        FuUnicodeCodepointCaseConvert := 43900;
        RETURN;
    5037:
        FuUnicodeCodepointCaseConvert := 43901;
        RETURN;
    5038:
        FuUnicodeCodepointCaseConvert := 43902;
        RETURN;
    5039:
        FuUnicodeCodepointCaseConvert := 43903;
        RETURN;
    5040:
        FuUnicodeCodepointCaseConvert := 43904;
        RETURN;
    5041:
        FuUnicodeCodepointCaseConvert := 43905;
        RETURN;
    5042:
        FuUnicodeCodepointCaseConvert := 43906;
        RETURN;
    5043:
        FuUnicodeCodepointCaseConvert := 43907;
        RETURN;
    5044:
        FuUnicodeCodepointCaseConvert := 43908;
        RETURN;
    5045:
        FuUnicodeCodepointCaseConvert := 43909;
        RETURN;
    5046:
        FuUnicodeCodepointCaseConvert := 43910;
        RETURN;
    5047:
        FuUnicodeCodepointCaseConvert := 43911;
        RETURN;
    5048:
        FuUnicodeCodepointCaseConvert := 43912;
        RETURN;
    5049:
        FuUnicodeCodepointCaseConvert := 43913;
        RETURN;
    5050:
        FuUnicodeCodepointCaseConvert := 43914;
        RETURN;
    5051:
        FuUnicodeCodepointCaseConvert := 43915;
        RETURN;
    5052:
        FuUnicodeCodepointCaseConvert := 43916;
        RETURN;
    5053:
        FuUnicodeCodepointCaseConvert := 43917;
        RETURN;
    5054:
        FuUnicodeCodepointCaseConvert := 43918;
        RETURN;
    5055:
        FuUnicodeCodepointCaseConvert := 43919;
        RETURN;
    5056:
        FuUnicodeCodepointCaseConvert := 43920;
        RETURN;
    5057:
        FuUnicodeCodepointCaseConvert := 43921;
        RETURN;
    5058:
        FuUnicodeCodepointCaseConvert := 43922;
        RETURN;
    5059:
        FuUnicodeCodepointCaseConvert := 43923;
        RETURN;
    5060:
        FuUnicodeCodepointCaseConvert := 43924;
        RETURN;
    5061:
        FuUnicodeCodepointCaseConvert := 43925;
        RETURN;
    5062:
        FuUnicodeCodepointCaseConvert := 43926;
        RETURN;
    5063:
        FuUnicodeCodepointCaseConvert := 43927;
        RETURN;
    5064:
        FuUnicodeCodepointCaseConvert := 43928;
        RETURN;
    5065:
        FuUnicodeCodepointCaseConvert := 43929;
        RETURN;
    5066:
        FuUnicodeCodepointCaseConvert := 43930;
        RETURN;
    5067:
        FuUnicodeCodepointCaseConvert := 43931;
        RETURN;
    5068:
        FuUnicodeCodepointCaseConvert := 43932;
        RETURN;
    5069:
        FuUnicodeCodepointCaseConvert := 43933;
        RETURN;
    5070:
        FuUnicodeCodepointCaseConvert := 43934;
        RETURN;
    5071:
        FuUnicodeCodepointCaseConvert := 43935;
        RETURN;
    5072:
        FuUnicodeCodepointCaseConvert := 43936;
        RETURN;
    5073:
        FuUnicodeCodepointCaseConvert := 43937;
        RETURN;
    5074:
        FuUnicodeCodepointCaseConvert := 43938;
        RETURN;
    5075:
        FuUnicodeCodepointCaseConvert := 43939;
        RETURN;
    5076:
        FuUnicodeCodepointCaseConvert := 43940;
        RETURN;
    5077:
        FuUnicodeCodepointCaseConvert := 43941;
        RETURN;
    5078:
        FuUnicodeCodepointCaseConvert := 43942;
        RETURN;
    5079:
        FuUnicodeCodepointCaseConvert := 43943;
        RETURN;
    5080:
        FuUnicodeCodepointCaseConvert := 43944;
        RETURN;
    5081:
        FuUnicodeCodepointCaseConvert := 43945;
        RETURN;
    5082:
        FuUnicodeCodepointCaseConvert := 43946;
        RETURN;
    5083:
        FuUnicodeCodepointCaseConvert := 43947;
        RETURN;
    5084:
        FuUnicodeCodepointCaseConvert := 43948;
        RETURN;
    5085:
        FuUnicodeCodepointCaseConvert := 43949;
        RETURN;
    5086:
        FuUnicodeCodepointCaseConvert := 43950;
        RETURN;
    5087:
        FuUnicodeCodepointCaseConvert := 43951;
        RETURN;
    5088:
        FuUnicodeCodepointCaseConvert := 43952;
        RETURN;
    5089:
        FuUnicodeCodepointCaseConvert := 43953;
        RETURN;
    5090:
        FuUnicodeCodepointCaseConvert := 43954;
        RETURN;
    5091:
        FuUnicodeCodepointCaseConvert := 43955;
        RETURN;
    5092:
        FuUnicodeCodepointCaseConvert := 43956;
        RETURN;
    5093:
        FuUnicodeCodepointCaseConvert := 43957;
        RETURN;
    5094:
        FuUnicodeCodepointCaseConvert := 43958;
        RETURN;
    5095:
        FuUnicodeCodepointCaseConvert := 43959;
        RETURN;
    5096:
        FuUnicodeCodepointCaseConvert := 43960;
        RETURN;
    5097:
        FuUnicodeCodepointCaseConvert := 43961;
        RETURN;
    5098:
        FuUnicodeCodepointCaseConvert := 43962;
        RETURN;
    5099:
        FuUnicodeCodepointCaseConvert := 43963;
        RETURN;
    5100:
        FuUnicodeCodepointCaseConvert := 43964;
        RETURN;
    5101:
        FuUnicodeCodepointCaseConvert := 43965;
        RETURN;
    5102:
        FuUnicodeCodepointCaseConvert := 43966;
        RETURN;
    5103:
        FuUnicodeCodepointCaseConvert := 43967;
        RETURN;
    5104:
        FuUnicodeCodepointCaseConvert := 5112;
        RETURN;
    5105:
        FuUnicodeCodepointCaseConvert := 5113;
        RETURN;
    5106:
        FuUnicodeCodepointCaseConvert := 5114;
        RETURN;
    5107:
        FuUnicodeCodepointCaseConvert := 5115;
        RETURN;
    5108:
        FuUnicodeCodepointCaseConvert := 5116;
        RETURN;
    5109:
        FuUnicodeCodepointCaseConvert := 5117;
        RETURN;
    5112:
        FuUnicodeCodepointCaseConvert := 5104;
        RETURN;
    5113:
        FuUnicodeCodepointCaseConvert := 5105;
        RETURN;
    5114:
        FuUnicodeCodepointCaseConvert := 5106;
        RETURN;
    5115:
        FuUnicodeCodepointCaseConvert := 5107;
        RETURN;
    5116:
        FuUnicodeCodepointCaseConvert := 5108;
        RETURN;
    5117:
        FuUnicodeCodepointCaseConvert := 5109;
        RETURN;
    7296:
        FuUnicodeCodepointCaseConvert := 1042;
        RETURN;
    7297:
        FuUnicodeCodepointCaseConvert := 1044;
        RETURN;
    7298:
        FuUnicodeCodepointCaseConvert := 1054;
        RETURN;
    7299:
        FuUnicodeCodepointCaseConvert := 1057;
        RETURN;
    7300:
        FuUnicodeCodepointCaseConvert := 1058;
        RETURN;
    7301:
        FuUnicodeCodepointCaseConvert := 1058;
        RETURN;
    7302:
        FuUnicodeCodepointCaseConvert := 1066;
        RETURN;
    7303:
        FuUnicodeCodepointCaseConvert := 1122;
        RETURN;
    7304:
        FuUnicodeCodepointCaseConvert := 42570;
        RETURN;
    7312:
        FuUnicodeCodepointCaseConvert := 4304;
        RETURN;
    7313:
        FuUnicodeCodepointCaseConvert := 4305;
        RETURN;
    7314:
        FuUnicodeCodepointCaseConvert := 4306;
        RETURN;
    7315:
        FuUnicodeCodepointCaseConvert := 4307;
        RETURN;
    7316:
        FuUnicodeCodepointCaseConvert := 4308;
        RETURN;
    7317:
        FuUnicodeCodepointCaseConvert := 4309;
        RETURN;
    7318:
        FuUnicodeCodepointCaseConvert := 4310;
        RETURN;
    7319:
        FuUnicodeCodepointCaseConvert := 4311;
        RETURN;
    7320:
        FuUnicodeCodepointCaseConvert := 4312;
        RETURN;
    7321:
        FuUnicodeCodepointCaseConvert := 4313;
        RETURN;
    7322:
        FuUnicodeCodepointCaseConvert := 4314;
        RETURN;
    7323:
        FuUnicodeCodepointCaseConvert := 4315;
        RETURN;
    7324:
        FuUnicodeCodepointCaseConvert := 4316;
        RETURN;
    7325:
        FuUnicodeCodepointCaseConvert := 4317;
        RETURN;
    7326:
        FuUnicodeCodepointCaseConvert := 4318;
        RETURN;
    7327:
        FuUnicodeCodepointCaseConvert := 4319;
        RETURN;
    7328:
        FuUnicodeCodepointCaseConvert := 4320;
        RETURN;
    7329:
        FuUnicodeCodepointCaseConvert := 4321;
        RETURN;
    7330:
        FuUnicodeCodepointCaseConvert := 4322;
        RETURN;
    7331:
        FuUnicodeCodepointCaseConvert := 4323;
        RETURN;
    7332:
        FuUnicodeCodepointCaseConvert := 4324;
        RETURN;
    7333:
        FuUnicodeCodepointCaseConvert := 4325;
        RETURN;
    7334:
        FuUnicodeCodepointCaseConvert := 4326;
        RETURN;
    7335:
        FuUnicodeCodepointCaseConvert := 4327;
        RETURN;
    7336:
        FuUnicodeCodepointCaseConvert := 4328;
        RETURN;
    7337:
        FuUnicodeCodepointCaseConvert := 4329;
        RETURN;
    7338:
        FuUnicodeCodepointCaseConvert := 4330;
        RETURN;
    7339:
        FuUnicodeCodepointCaseConvert := 4331;
        RETURN;
    7340:
        FuUnicodeCodepointCaseConvert := 4332;
        RETURN;
    7341:
        FuUnicodeCodepointCaseConvert := 4333;
        RETURN;
    7342:
        FuUnicodeCodepointCaseConvert := 4334;
        RETURN;
    7343:
        FuUnicodeCodepointCaseConvert := 4335;
        RETURN;
    7344:
        FuUnicodeCodepointCaseConvert := 4336;
        RETURN;
    7345:
        FuUnicodeCodepointCaseConvert := 4337;
        RETURN;
    7346:
        FuUnicodeCodepointCaseConvert := 4338;
        RETURN;
    7347:
        FuUnicodeCodepointCaseConvert := 4339;
        RETURN;
    7348:
        FuUnicodeCodepointCaseConvert := 4340;
        RETURN;
    7349:
        FuUnicodeCodepointCaseConvert := 4341;
        RETURN;
    7350:
        FuUnicodeCodepointCaseConvert := 4342;
        RETURN;
    7351:
        FuUnicodeCodepointCaseConvert := 4343;
        RETURN;
    7352:
        FuUnicodeCodepointCaseConvert := 4344;
        RETURN;
    7353:
        FuUnicodeCodepointCaseConvert := 4345;
        RETURN;
    7354:
        FuUnicodeCodepointCaseConvert := 4346;
        RETURN;
    7357:
        FuUnicodeCodepointCaseConvert := 4349;
        RETURN;
    7358:
        FuUnicodeCodepointCaseConvert := 4350;
        RETURN;
    7359:
        FuUnicodeCodepointCaseConvert := 4351;
        RETURN;
    7545:
        FuUnicodeCodepointCaseConvert := 42877;
        RETURN;
    7549:
        FuUnicodeCodepointCaseConvert := 11363;
        RETURN;
    7566:
        FuUnicodeCodepointCaseConvert := 42950;
        RETURN;
    7680:
        FuUnicodeCodepointCaseConvert := 7681;
        RETURN;
    7681:
        FuUnicodeCodepointCaseConvert := 7680;
        RETURN;
    7682:
        FuUnicodeCodepointCaseConvert := 7683;
        RETURN;
    7683:
        FuUnicodeCodepointCaseConvert := 7682;
        RETURN;
    7684:
        FuUnicodeCodepointCaseConvert := 7685;
        RETURN;
    7685:
        FuUnicodeCodepointCaseConvert := 7684;
        RETURN;
    7686:
        FuUnicodeCodepointCaseConvert := 7687;
        RETURN;
    7687:
        FuUnicodeCodepointCaseConvert := 7686;
        RETURN;
    7688:
        FuUnicodeCodepointCaseConvert := 7689;
        RETURN;
    7689:
        FuUnicodeCodepointCaseConvert := 7688;
        RETURN;
    7690:
        FuUnicodeCodepointCaseConvert := 7691;
        RETURN;
    7691:
        FuUnicodeCodepointCaseConvert := 7690;
        RETURN;
    7692:
        FuUnicodeCodepointCaseConvert := 7693;
        RETURN;
    7693:
        FuUnicodeCodepointCaseConvert := 7692;
        RETURN;
    7694:
        FuUnicodeCodepointCaseConvert := 7695;
        RETURN;
    7695:
        FuUnicodeCodepointCaseConvert := 7694;
        RETURN;
    7696:
        FuUnicodeCodepointCaseConvert := 7697;
        RETURN;
    7697:
        FuUnicodeCodepointCaseConvert := 7696;
        RETURN;
    7698:
        FuUnicodeCodepointCaseConvert := 7699;
        RETURN;
    7699:
        FuUnicodeCodepointCaseConvert := 7698;
        RETURN;
    7700:
        FuUnicodeCodepointCaseConvert := 7701;
        RETURN;
    7701:
        FuUnicodeCodepointCaseConvert := 7700;
        RETURN;
    7702:
        FuUnicodeCodepointCaseConvert := 7703;
        RETURN;
    7703:
        FuUnicodeCodepointCaseConvert := 7702;
        RETURN;
    7704:
        FuUnicodeCodepointCaseConvert := 7705;
        RETURN;
    7705:
        FuUnicodeCodepointCaseConvert := 7704;
        RETURN;
    7706:
        FuUnicodeCodepointCaseConvert := 7707;
        RETURN;
    7707:
        FuUnicodeCodepointCaseConvert := 7706;
        RETURN;
    7708:
        FuUnicodeCodepointCaseConvert := 7709;
        RETURN;
    7709:
        FuUnicodeCodepointCaseConvert := 7708;
        RETURN;
    7710:
        FuUnicodeCodepointCaseConvert := 7711;
        RETURN;
    7711:
        FuUnicodeCodepointCaseConvert := 7710;
        RETURN;
    7712:
        FuUnicodeCodepointCaseConvert := 7713;
        RETURN;
    7713:
        FuUnicodeCodepointCaseConvert := 7712;
        RETURN;
    7714:
        FuUnicodeCodepointCaseConvert := 7715;
        RETURN;
    7715:
        FuUnicodeCodepointCaseConvert := 7714;
        RETURN;
    7716:
        FuUnicodeCodepointCaseConvert := 7717;
        RETURN;
    7717:
        FuUnicodeCodepointCaseConvert := 7716;
        RETURN;
    7718:
        FuUnicodeCodepointCaseConvert := 7719;
        RETURN;
    7719:
        FuUnicodeCodepointCaseConvert := 7718;
        RETURN;
    7720:
        FuUnicodeCodepointCaseConvert := 7721;
        RETURN;
    7721:
        FuUnicodeCodepointCaseConvert := 7720;
        RETURN;
    7722:
        FuUnicodeCodepointCaseConvert := 7723;
        RETURN;
    7723:
        FuUnicodeCodepointCaseConvert := 7722;
        RETURN;
    7724:
        FuUnicodeCodepointCaseConvert := 7725;
        RETURN;
    7725:
        FuUnicodeCodepointCaseConvert := 7724;
        RETURN;
    7726:
        FuUnicodeCodepointCaseConvert := 7727;
        RETURN;
    7727:
        FuUnicodeCodepointCaseConvert := 7726;
        RETURN;
    7728:
        FuUnicodeCodepointCaseConvert := 7729;
        RETURN;
    7729:
        FuUnicodeCodepointCaseConvert := 7728;
        RETURN;
    7730:
        FuUnicodeCodepointCaseConvert := 7731;
        RETURN;
    7731:
        FuUnicodeCodepointCaseConvert := 7730;
        RETURN;
    7732:
        FuUnicodeCodepointCaseConvert := 7733;
        RETURN;
    7733:
        FuUnicodeCodepointCaseConvert := 7732;
        RETURN;
    7734:
        FuUnicodeCodepointCaseConvert := 7735;
        RETURN;
    7735:
        FuUnicodeCodepointCaseConvert := 7734;
        RETURN;
    7736:
        FuUnicodeCodepointCaseConvert := 7737;
        RETURN;
    7737:
        FuUnicodeCodepointCaseConvert := 7736;
        RETURN;
    7738:
        FuUnicodeCodepointCaseConvert := 7739;
        RETURN;
    7739:
        FuUnicodeCodepointCaseConvert := 7738;
        RETURN;
    7740:
        FuUnicodeCodepointCaseConvert := 7741;
        RETURN;
    7741:
        FuUnicodeCodepointCaseConvert := 7740;
        RETURN;
    7742:
        FuUnicodeCodepointCaseConvert := 7743;
        RETURN;
    7743:
        FuUnicodeCodepointCaseConvert := 7742;
        RETURN;
    7744:
        FuUnicodeCodepointCaseConvert := 7745;
        RETURN;
    7745:
        FuUnicodeCodepointCaseConvert := 7744;
        RETURN;
    7746:
        FuUnicodeCodepointCaseConvert := 7747;
        RETURN;
    7747:
        FuUnicodeCodepointCaseConvert := 7746;
        RETURN;
    7748:
        FuUnicodeCodepointCaseConvert := 7749;
        RETURN;
    7749:
        FuUnicodeCodepointCaseConvert := 7748;
        RETURN;
    7750:
        FuUnicodeCodepointCaseConvert := 7751;
        RETURN;
    7751:
        FuUnicodeCodepointCaseConvert := 7750;
        RETURN;
    7752:
        FuUnicodeCodepointCaseConvert := 7753;
        RETURN;
    7753:
        FuUnicodeCodepointCaseConvert := 7752;
        RETURN;
    7754:
        FuUnicodeCodepointCaseConvert := 7755;
        RETURN;
    7755:
        FuUnicodeCodepointCaseConvert := 7754;
        RETURN;
    7756:
        FuUnicodeCodepointCaseConvert := 7757;
        RETURN;
    7757:
        FuUnicodeCodepointCaseConvert := 7756;
        RETURN;
    7758:
        FuUnicodeCodepointCaseConvert := 7759;
        RETURN;
    7759:
        FuUnicodeCodepointCaseConvert := 7758;
        RETURN;
    7760:
        FuUnicodeCodepointCaseConvert := 7761;
        RETURN;
    7761:
        FuUnicodeCodepointCaseConvert := 7760;
        RETURN;
    7762:
        FuUnicodeCodepointCaseConvert := 7763;
        RETURN;
    7763:
        FuUnicodeCodepointCaseConvert := 7762;
        RETURN;
    7764:
        FuUnicodeCodepointCaseConvert := 7765;
        RETURN;
    7765:
        FuUnicodeCodepointCaseConvert := 7764;
        RETURN;
    7766:
        FuUnicodeCodepointCaseConvert := 7767;
        RETURN;
    7767:
        FuUnicodeCodepointCaseConvert := 7766;
        RETURN;
    7768:
        FuUnicodeCodepointCaseConvert := 7769;
        RETURN;
    7769:
        FuUnicodeCodepointCaseConvert := 7768;
        RETURN;
    7770:
        FuUnicodeCodepointCaseConvert := 7771;
        RETURN;
    7771:
        FuUnicodeCodepointCaseConvert := 7770;
        RETURN;
    7772:
        FuUnicodeCodepointCaseConvert := 7773;
        RETURN;
    7773:
        FuUnicodeCodepointCaseConvert := 7772;
        RETURN;
    7774:
        FuUnicodeCodepointCaseConvert := 7775;
        RETURN;
    7775:
        FuUnicodeCodepointCaseConvert := 7774;
        RETURN;
    7776:
        FuUnicodeCodepointCaseConvert := 7777;
        RETURN;
    7777:
        FuUnicodeCodepointCaseConvert := 7776;
        RETURN;
    7778:
        FuUnicodeCodepointCaseConvert := 7779;
        RETURN;
    7779:
        FuUnicodeCodepointCaseConvert := 7778;
        RETURN;
    7780:
        FuUnicodeCodepointCaseConvert := 7781;
        RETURN;
    7781:
        FuUnicodeCodepointCaseConvert := 7780;
        RETURN;
    7782:
        FuUnicodeCodepointCaseConvert := 7783;
        RETURN;
    7783:
        FuUnicodeCodepointCaseConvert := 7782;
        RETURN;
    7784:
        FuUnicodeCodepointCaseConvert := 7785;
        RETURN;
    7785:
        FuUnicodeCodepointCaseConvert := 7784;
        RETURN;
    7786:
        FuUnicodeCodepointCaseConvert := 7787;
        RETURN;
    7787:
        FuUnicodeCodepointCaseConvert := 7786;
        RETURN;
    7788:
        FuUnicodeCodepointCaseConvert := 7789;
        RETURN;
    7789:
        FuUnicodeCodepointCaseConvert := 7788;
        RETURN;
    7790:
        FuUnicodeCodepointCaseConvert := 7791;
        RETURN;
    7791:
        FuUnicodeCodepointCaseConvert := 7790;
        RETURN;
    7792:
        FuUnicodeCodepointCaseConvert := 7793;
        RETURN;
    7793:
        FuUnicodeCodepointCaseConvert := 7792;
        RETURN;
    7794:
        FuUnicodeCodepointCaseConvert := 7795;
        RETURN;
    7795:
        FuUnicodeCodepointCaseConvert := 7794;
        RETURN;
    7796:
        FuUnicodeCodepointCaseConvert := 7797;
        RETURN;
    7797:
        FuUnicodeCodepointCaseConvert := 7796;
        RETURN;
    7798:
        FuUnicodeCodepointCaseConvert := 7799;
        RETURN;
    7799:
        FuUnicodeCodepointCaseConvert := 7798;
        RETURN;
    7800:
        FuUnicodeCodepointCaseConvert := 7801;
        RETURN;
    7801:
        FuUnicodeCodepointCaseConvert := 7800;
        RETURN;
    7802:
        FuUnicodeCodepointCaseConvert := 7803;
        RETURN;
    7803:
        FuUnicodeCodepointCaseConvert := 7802;
        RETURN;
    7804:
        FuUnicodeCodepointCaseConvert := 7805;
        RETURN;
    7805:
        FuUnicodeCodepointCaseConvert := 7804;
        RETURN;
    7806:
        FuUnicodeCodepointCaseConvert := 7807;
        RETURN;
    7807:
        FuUnicodeCodepointCaseConvert := 7806;
        RETURN;
    7808:
        FuUnicodeCodepointCaseConvert := 7809;
        RETURN;
    7809:
        FuUnicodeCodepointCaseConvert := 7808;
        RETURN;
    7810:
        FuUnicodeCodepointCaseConvert := 7811;
        RETURN;
    7811:
        FuUnicodeCodepointCaseConvert := 7810;
        RETURN;
    7812:
        FuUnicodeCodepointCaseConvert := 7813;
        RETURN;
    7813:
        FuUnicodeCodepointCaseConvert := 7812;
        RETURN;
    7814:
        FuUnicodeCodepointCaseConvert := 7815;
        RETURN;
    7815:
        FuUnicodeCodepointCaseConvert := 7814;
        RETURN;
    7816:
        FuUnicodeCodepointCaseConvert := 7817;
        RETURN;
    7817:
        FuUnicodeCodepointCaseConvert := 7816;
        RETURN;
    7818:
        FuUnicodeCodepointCaseConvert := 7819;
        RETURN;
    7819:
        FuUnicodeCodepointCaseConvert := 7818;
        RETURN;
    7820:
        FuUnicodeCodepointCaseConvert := 7821;
        RETURN;
    7821:
        FuUnicodeCodepointCaseConvert := 7820;
        RETURN;
    7822:
        FuUnicodeCodepointCaseConvert := 7823;
        RETURN;
    7823:
        FuUnicodeCodepointCaseConvert := 7822;
        RETURN;
    7824:
        FuUnicodeCodepointCaseConvert := 7825;
        RETURN;
    7825:
        FuUnicodeCodepointCaseConvert := 7824;
        RETURN;
    7826:
        FuUnicodeCodepointCaseConvert := 7827;
        RETURN;
    7827:
        FuUnicodeCodepointCaseConvert := 7826;
        RETURN;
    7828:
        FuUnicodeCodepointCaseConvert := 7829;
        RETURN;
    7829:
        FuUnicodeCodepointCaseConvert := 7828;
        RETURN;
    7835:
        FuUnicodeCodepointCaseConvert := 7776;
        RETURN;
    7838:
        FuUnicodeCodepointCaseConvert := 223;
        RETURN;
    7840:
        FuUnicodeCodepointCaseConvert := 7841;
        RETURN;
    7841:
        FuUnicodeCodepointCaseConvert := 7840;
        RETURN;
    7842:
        FuUnicodeCodepointCaseConvert := 7843;
        RETURN;
    7843:
        FuUnicodeCodepointCaseConvert := 7842;
        RETURN;
    7844:
        FuUnicodeCodepointCaseConvert := 7845;
        RETURN;
    7845:
        FuUnicodeCodepointCaseConvert := 7844;
        RETURN;
    7846:
        FuUnicodeCodepointCaseConvert := 7847;
        RETURN;
    7847:
        FuUnicodeCodepointCaseConvert := 7846;
        RETURN;
    7848:
        FuUnicodeCodepointCaseConvert := 7849;
        RETURN;
    7849:
        FuUnicodeCodepointCaseConvert := 7848;
        RETURN;
    7850:
        FuUnicodeCodepointCaseConvert := 7851;
        RETURN;
    7851:
        FuUnicodeCodepointCaseConvert := 7850;
        RETURN;
    7852:
        FuUnicodeCodepointCaseConvert := 7853;
        RETURN;
    7853:
        FuUnicodeCodepointCaseConvert := 7852;
        RETURN;
    7854:
        FuUnicodeCodepointCaseConvert := 7855;
        RETURN;
    7855:
        FuUnicodeCodepointCaseConvert := 7854;
        RETURN;
    7856:
        FuUnicodeCodepointCaseConvert := 7857;
        RETURN;
    7857:
        FuUnicodeCodepointCaseConvert := 7856;
        RETURN;
    7858:
        FuUnicodeCodepointCaseConvert := 7859;
        RETURN;
    7859:
        FuUnicodeCodepointCaseConvert := 7858;
        RETURN;
    7860:
        FuUnicodeCodepointCaseConvert := 7861;
        RETURN;
    7861:
        FuUnicodeCodepointCaseConvert := 7860;
        RETURN;
    7862:
        FuUnicodeCodepointCaseConvert := 7863;
        RETURN;
    7863:
        FuUnicodeCodepointCaseConvert := 7862;
        RETURN;
    7864:
        FuUnicodeCodepointCaseConvert := 7865;
        RETURN;
    7865:
        FuUnicodeCodepointCaseConvert := 7864;
        RETURN;
    7866:
        FuUnicodeCodepointCaseConvert := 7867;
        RETURN;
    7867:
        FuUnicodeCodepointCaseConvert := 7866;
        RETURN;
    7868:
        FuUnicodeCodepointCaseConvert := 7869;
        RETURN;
    7869:
        FuUnicodeCodepointCaseConvert := 7868;
        RETURN;
    7870:
        FuUnicodeCodepointCaseConvert := 7871;
        RETURN;
    7871:
        FuUnicodeCodepointCaseConvert := 7870;
        RETURN;
    7872:
        FuUnicodeCodepointCaseConvert := 7873;
        RETURN;
    7873:
        FuUnicodeCodepointCaseConvert := 7872;
        RETURN;
    7874:
        FuUnicodeCodepointCaseConvert := 7875;
        RETURN;
    7875:
        FuUnicodeCodepointCaseConvert := 7874;
        RETURN;
    7876:
        FuUnicodeCodepointCaseConvert := 7877;
        RETURN;
    7877:
        FuUnicodeCodepointCaseConvert := 7876;
        RETURN;
    7878:
        FuUnicodeCodepointCaseConvert := 7879;
        RETURN;
    7879:
        FuUnicodeCodepointCaseConvert := 7878;
        RETURN;
    7880:
        FuUnicodeCodepointCaseConvert := 7881;
        RETURN;
    7881:
        FuUnicodeCodepointCaseConvert := 7880;
        RETURN;
    7882:
        FuUnicodeCodepointCaseConvert := 7883;
        RETURN;
    7883:
        FuUnicodeCodepointCaseConvert := 7882;
        RETURN;
    7884:
        FuUnicodeCodepointCaseConvert := 7885;
        RETURN;
    7885:
        FuUnicodeCodepointCaseConvert := 7884;
        RETURN;
    7886:
        FuUnicodeCodepointCaseConvert := 7887;
        RETURN;
    7887:
        FuUnicodeCodepointCaseConvert := 7886;
        RETURN;
    7888:
        FuUnicodeCodepointCaseConvert := 7889;
        RETURN;
    7889:
        FuUnicodeCodepointCaseConvert := 7888;
        RETURN;
    7890:
        FuUnicodeCodepointCaseConvert := 7891;
        RETURN;
    7891:
        FuUnicodeCodepointCaseConvert := 7890;
        RETURN;
    7892:
        FuUnicodeCodepointCaseConvert := 7893;
        RETURN;
    7893:
        FuUnicodeCodepointCaseConvert := 7892;
        RETURN;
    7894:
        FuUnicodeCodepointCaseConvert := 7895;
        RETURN;
    7895:
        FuUnicodeCodepointCaseConvert := 7894;
        RETURN;
    7896:
        FuUnicodeCodepointCaseConvert := 7897;
        RETURN;
    7897:
        FuUnicodeCodepointCaseConvert := 7896;
        RETURN;
    7898:
        FuUnicodeCodepointCaseConvert := 7899;
        RETURN;
    7899:
        FuUnicodeCodepointCaseConvert := 7898;
        RETURN;
    7900:
        FuUnicodeCodepointCaseConvert := 7901;
        RETURN;
    7901:
        FuUnicodeCodepointCaseConvert := 7900;
        RETURN;
    7902:
        FuUnicodeCodepointCaseConvert := 7903;
        RETURN;
    7903:
        FuUnicodeCodepointCaseConvert := 7902;
        RETURN;
    7904:
        FuUnicodeCodepointCaseConvert := 7905;
        RETURN;
    7905:
        FuUnicodeCodepointCaseConvert := 7904;
        RETURN;
    7906:
        FuUnicodeCodepointCaseConvert := 7907;
        RETURN;
    7907:
        FuUnicodeCodepointCaseConvert := 7906;
        RETURN;
    7908:
        FuUnicodeCodepointCaseConvert := 7909;
        RETURN;
    7909:
        FuUnicodeCodepointCaseConvert := 7908;
        RETURN;
    7910:
        FuUnicodeCodepointCaseConvert := 7911;
        RETURN;
    7911:
        FuUnicodeCodepointCaseConvert := 7910;
        RETURN;
    7912:
        FuUnicodeCodepointCaseConvert := 7913;
        RETURN;
    7913:
        FuUnicodeCodepointCaseConvert := 7912;
        RETURN;
    7914:
        FuUnicodeCodepointCaseConvert := 7915;
        RETURN;
    7915:
        FuUnicodeCodepointCaseConvert := 7914;
        RETURN;
    7916:
        FuUnicodeCodepointCaseConvert := 7917;
        RETURN;
    7917:
        FuUnicodeCodepointCaseConvert := 7916;
        RETURN;
    7918:
        FuUnicodeCodepointCaseConvert := 7919;
        RETURN;
    7919:
        FuUnicodeCodepointCaseConvert := 7918;
        RETURN;
    7920:
        FuUnicodeCodepointCaseConvert := 7921;
        RETURN;
    7921:
        FuUnicodeCodepointCaseConvert := 7920;
        RETURN;
    7922:
        FuUnicodeCodepointCaseConvert := 7923;
        RETURN;
    7923:
        FuUnicodeCodepointCaseConvert := 7922;
        RETURN;
    7924:
        FuUnicodeCodepointCaseConvert := 7925;
        RETURN;
    7925:
        FuUnicodeCodepointCaseConvert := 7924;
        RETURN;
    7926:
        FuUnicodeCodepointCaseConvert := 7927;
        RETURN;
    7927:
        FuUnicodeCodepointCaseConvert := 7926;
        RETURN;
    7928:
        FuUnicodeCodepointCaseConvert := 7929;
        RETURN;
    7929:
        FuUnicodeCodepointCaseConvert := 7928;
        RETURN;
    7930:
        FuUnicodeCodepointCaseConvert := 7931;
        RETURN;
    7931:
        FuUnicodeCodepointCaseConvert := 7930;
        RETURN;
    7932:
        FuUnicodeCodepointCaseConvert := 7933;
        RETURN;
    7933:
        FuUnicodeCodepointCaseConvert := 7932;
        RETURN;
    7934:
        FuUnicodeCodepointCaseConvert := 7935;
        RETURN;
    7935:
        FuUnicodeCodepointCaseConvert := 7934;
        RETURN;
    7936:
        FuUnicodeCodepointCaseConvert := 7944;
        RETURN;
    7937:
        FuUnicodeCodepointCaseConvert := 7945;
        RETURN;
    7938:
        FuUnicodeCodepointCaseConvert := 7946;
        RETURN;
    7939:
        FuUnicodeCodepointCaseConvert := 7947;
        RETURN;
    7940:
        FuUnicodeCodepointCaseConvert := 7948;
        RETURN;
    7941:
        FuUnicodeCodepointCaseConvert := 7949;
        RETURN;
    7942:
        FuUnicodeCodepointCaseConvert := 7950;
        RETURN;
    7943:
        FuUnicodeCodepointCaseConvert := 7951;
        RETURN;
    7944:
        FuUnicodeCodepointCaseConvert := 7936;
        RETURN;
    7945:
        FuUnicodeCodepointCaseConvert := 7937;
        RETURN;
    7946:
        FuUnicodeCodepointCaseConvert := 7938;
        RETURN;
    7947:
        FuUnicodeCodepointCaseConvert := 7939;
        RETURN;
    7948:
        FuUnicodeCodepointCaseConvert := 7940;
        RETURN;
    7949:
        FuUnicodeCodepointCaseConvert := 7941;
        RETURN;
    7950:
        FuUnicodeCodepointCaseConvert := 7942;
        RETURN;
    7951:
        FuUnicodeCodepointCaseConvert := 7943;
        RETURN;
    7952:
        FuUnicodeCodepointCaseConvert := 7960;
        RETURN;
    7953:
        FuUnicodeCodepointCaseConvert := 7961;
        RETURN;
    7954:
        FuUnicodeCodepointCaseConvert := 7962;
        RETURN;
    7955:
        FuUnicodeCodepointCaseConvert := 7963;
        RETURN;
    7956:
        FuUnicodeCodepointCaseConvert := 7964;
        RETURN;
    7957:
        FuUnicodeCodepointCaseConvert := 7965;
        RETURN;
    7960:
        FuUnicodeCodepointCaseConvert := 7952;
        RETURN;
    7961:
        FuUnicodeCodepointCaseConvert := 7953;
        RETURN;
    7962:
        FuUnicodeCodepointCaseConvert := 7954;
        RETURN;
    7963:
        FuUnicodeCodepointCaseConvert := 7955;
        RETURN;
    7964:
        FuUnicodeCodepointCaseConvert := 7956;
        RETURN;
    7965:
        FuUnicodeCodepointCaseConvert := 7957;
        RETURN;
    7968:
        FuUnicodeCodepointCaseConvert := 7976;
        RETURN;
    7969:
        FuUnicodeCodepointCaseConvert := 7977;
        RETURN;
    7970:
        FuUnicodeCodepointCaseConvert := 7978;
        RETURN;
    7971:
        FuUnicodeCodepointCaseConvert := 7979;
        RETURN;
    7972:
        FuUnicodeCodepointCaseConvert := 7980;
        RETURN;
    7973:
        FuUnicodeCodepointCaseConvert := 7981;
        RETURN;
    7974:
        FuUnicodeCodepointCaseConvert := 7982;
        RETURN;
    7975:
        FuUnicodeCodepointCaseConvert := 7983;
        RETURN;
    7976:
        FuUnicodeCodepointCaseConvert := 7968;
        RETURN;
    7977:
        FuUnicodeCodepointCaseConvert := 7969;
        RETURN;
    7978:
        FuUnicodeCodepointCaseConvert := 7970;
        RETURN;
    7979:
        FuUnicodeCodepointCaseConvert := 7971;
        RETURN;
    7980:
        FuUnicodeCodepointCaseConvert := 7972;
        RETURN;
    7981:
        FuUnicodeCodepointCaseConvert := 7973;
        RETURN;
    7982:
        FuUnicodeCodepointCaseConvert := 7974;
        RETURN;
    7983:
        FuUnicodeCodepointCaseConvert := 7975;
        RETURN;
    7984:
        FuUnicodeCodepointCaseConvert := 7992;
        RETURN;
    7985:
        FuUnicodeCodepointCaseConvert := 7993;
        RETURN;
    7986:
        FuUnicodeCodepointCaseConvert := 7994;
        RETURN;
    7987:
        FuUnicodeCodepointCaseConvert := 7995;
        RETURN;
    7988:
        FuUnicodeCodepointCaseConvert := 7996;
        RETURN;
    7989:
        FuUnicodeCodepointCaseConvert := 7997;
        RETURN;
    7990:
        FuUnicodeCodepointCaseConvert := 7998;
        RETURN;
    7991:
        FuUnicodeCodepointCaseConvert := 7999;
        RETURN;
    7992:
        FuUnicodeCodepointCaseConvert := 7984;
        RETURN;
    7993:
        FuUnicodeCodepointCaseConvert := 7985;
        RETURN;
    7994:
        FuUnicodeCodepointCaseConvert := 7986;
        RETURN;
    7995:
        FuUnicodeCodepointCaseConvert := 7987;
        RETURN;
    7996:
        FuUnicodeCodepointCaseConvert := 7988;
        RETURN;
    7997:
        FuUnicodeCodepointCaseConvert := 7989;
        RETURN;
    7998:
        FuUnicodeCodepointCaseConvert := 7990;
        RETURN;
    7999:
        FuUnicodeCodepointCaseConvert := 7991;
        RETURN;
    8000:
        FuUnicodeCodepointCaseConvert := 8008;
        RETURN;
    8001:
        FuUnicodeCodepointCaseConvert := 8009;
        RETURN;
    8002:
        FuUnicodeCodepointCaseConvert := 8010;
        RETURN;
    8003:
        FuUnicodeCodepointCaseConvert := 8011;
        RETURN;
    8004:
        FuUnicodeCodepointCaseConvert := 8012;
        RETURN;
    8005:
        FuUnicodeCodepointCaseConvert := 8013;
        RETURN;
    8008:
        FuUnicodeCodepointCaseConvert := 8000;
        RETURN;
    8009:
        FuUnicodeCodepointCaseConvert := 8001;
        RETURN;
    8010:
        FuUnicodeCodepointCaseConvert := 8002;
        RETURN;
    8011:
        FuUnicodeCodepointCaseConvert := 8003;
        RETURN;
    8012:
        FuUnicodeCodepointCaseConvert := 8004;
        RETURN;
    8013:
        FuUnicodeCodepointCaseConvert := 8005;
        RETURN;
    8017:
        FuUnicodeCodepointCaseConvert := 8025;
        RETURN;
    8019:
        FuUnicodeCodepointCaseConvert := 8027;
        RETURN;
    8021:
        FuUnicodeCodepointCaseConvert := 8029;
        RETURN;
    8023:
        FuUnicodeCodepointCaseConvert := 8031;
        RETURN;
    8025:
        FuUnicodeCodepointCaseConvert := 8017;
        RETURN;
    8027:
        FuUnicodeCodepointCaseConvert := 8019;
        RETURN;
    8029:
        FuUnicodeCodepointCaseConvert := 8021;
        RETURN;
    8031:
        FuUnicodeCodepointCaseConvert := 8023;
        RETURN;
    8032:
        FuUnicodeCodepointCaseConvert := 8040;
        RETURN;
    8033:
        FuUnicodeCodepointCaseConvert := 8041;
        RETURN;
    8034:
        FuUnicodeCodepointCaseConvert := 8042;
        RETURN;
    8035:
        FuUnicodeCodepointCaseConvert := 8043;
        RETURN;
    8036:
        FuUnicodeCodepointCaseConvert := 8044;
        RETURN;
    8037:
        FuUnicodeCodepointCaseConvert := 8045;
        RETURN;
    8038:
        FuUnicodeCodepointCaseConvert := 8046;
        RETURN;
    8039:
        FuUnicodeCodepointCaseConvert := 8047;
        RETURN;
    8040:
        FuUnicodeCodepointCaseConvert := 8032;
        RETURN;
    8041:
        FuUnicodeCodepointCaseConvert := 8033;
        RETURN;
    8042:
        FuUnicodeCodepointCaseConvert := 8034;
        RETURN;
    8043:
        FuUnicodeCodepointCaseConvert := 8035;
        RETURN;
    8044:
        FuUnicodeCodepointCaseConvert := 8036;
        RETURN;
    8045:
        FuUnicodeCodepointCaseConvert := 8037;
        RETURN;
    8046:
        FuUnicodeCodepointCaseConvert := 8038;
        RETURN;
    8047:
        FuUnicodeCodepointCaseConvert := 8039;
        RETURN;
    8048:
        FuUnicodeCodepointCaseConvert := 8122;
        RETURN;
    8049:
        FuUnicodeCodepointCaseConvert := 8123;
        RETURN;
    8050:
        FuUnicodeCodepointCaseConvert := 8136;
        RETURN;
    8051:
        FuUnicodeCodepointCaseConvert := 8137;
        RETURN;
    8052:
        FuUnicodeCodepointCaseConvert := 8138;
        RETURN;
    8053:
        FuUnicodeCodepointCaseConvert := 8139;
        RETURN;
    8054:
        FuUnicodeCodepointCaseConvert := 8154;
        RETURN;
    8055:
        FuUnicodeCodepointCaseConvert := 8155;
        RETURN;
    8056:
        FuUnicodeCodepointCaseConvert := 8184;
        RETURN;
    8057:
        FuUnicodeCodepointCaseConvert := 8185;
        RETURN;
    8058:
        FuUnicodeCodepointCaseConvert := 8170;
        RETURN;
    8059:
        FuUnicodeCodepointCaseConvert := 8171;
        RETURN;
    8060:
        FuUnicodeCodepointCaseConvert := 8186;
        RETURN;
    8061:
        FuUnicodeCodepointCaseConvert := 8187;
        RETURN;
    8064:
        FuUnicodeCodepointCaseConvert := 8072;
        RETURN;
    8065:
        FuUnicodeCodepointCaseConvert := 8073;
        RETURN;
    8066:
        FuUnicodeCodepointCaseConvert := 8074;
        RETURN;
    8067:
        FuUnicodeCodepointCaseConvert := 8075;
        RETURN;
    8068:
        FuUnicodeCodepointCaseConvert := 8076;
        RETURN;
    8069:
        FuUnicodeCodepointCaseConvert := 8077;
        RETURN;
    8070:
        FuUnicodeCodepointCaseConvert := 8078;
        RETURN;
    8071:
        FuUnicodeCodepointCaseConvert := 8079;
        RETURN;
    8072:
        FuUnicodeCodepointCaseConvert := 8064;
        RETURN;
    8073:
        FuUnicodeCodepointCaseConvert := 8065;
        RETURN;
    8074:
        FuUnicodeCodepointCaseConvert := 8066;
        RETURN;
    8075:
        FuUnicodeCodepointCaseConvert := 8067;
        RETURN;
    8076:
        FuUnicodeCodepointCaseConvert := 8068;
        RETURN;
    8077:
        FuUnicodeCodepointCaseConvert := 8069;
        RETURN;
    8078:
        FuUnicodeCodepointCaseConvert := 8070;
        RETURN;
    8079:
        FuUnicodeCodepointCaseConvert := 8071;
        RETURN;
    8080:
        FuUnicodeCodepointCaseConvert := 8088;
        RETURN;
    8081:
        FuUnicodeCodepointCaseConvert := 8089;
        RETURN;
    8082:
        FuUnicodeCodepointCaseConvert := 8090;
        RETURN;
    8083:
        FuUnicodeCodepointCaseConvert := 8091;
        RETURN;
    8084:
        FuUnicodeCodepointCaseConvert := 8092;
        RETURN;
    8085:
        FuUnicodeCodepointCaseConvert := 8093;
        RETURN;
    8086:
        FuUnicodeCodepointCaseConvert := 8094;
        RETURN;
    8087:
        FuUnicodeCodepointCaseConvert := 8095;
        RETURN;
    8088:
        FuUnicodeCodepointCaseConvert := 8080;
        RETURN;
    8089:
        FuUnicodeCodepointCaseConvert := 8081;
        RETURN;
    8090:
        FuUnicodeCodepointCaseConvert := 8082;
        RETURN;
    8091:
        FuUnicodeCodepointCaseConvert := 8083;
        RETURN;
    8092:
        FuUnicodeCodepointCaseConvert := 8084;
        RETURN;
    8093:
        FuUnicodeCodepointCaseConvert := 8085;
        RETURN;
    8094:
        FuUnicodeCodepointCaseConvert := 8086;
        RETURN;
    8095:
        FuUnicodeCodepointCaseConvert := 8087;
        RETURN;
    8096:
        FuUnicodeCodepointCaseConvert := 8104;
        RETURN;
    8097:
        FuUnicodeCodepointCaseConvert := 8105;
        RETURN;
    8098:
        FuUnicodeCodepointCaseConvert := 8106;
        RETURN;
    8099:
        FuUnicodeCodepointCaseConvert := 8107;
        RETURN;
    8100:
        FuUnicodeCodepointCaseConvert := 8108;
        RETURN;
    8101:
        FuUnicodeCodepointCaseConvert := 8109;
        RETURN;
    8102:
        FuUnicodeCodepointCaseConvert := 8110;
        RETURN;
    8103:
        FuUnicodeCodepointCaseConvert := 8111;
        RETURN;
    8104:
        FuUnicodeCodepointCaseConvert := 8096;
        RETURN;
    8105:
        FuUnicodeCodepointCaseConvert := 8097;
        RETURN;
    8106:
        FuUnicodeCodepointCaseConvert := 8098;
        RETURN;
    8107:
        FuUnicodeCodepointCaseConvert := 8099;
        RETURN;
    8108:
        FuUnicodeCodepointCaseConvert := 8100;
        RETURN;
    8109:
        FuUnicodeCodepointCaseConvert := 8101;
        RETURN;
    8110:
        FuUnicodeCodepointCaseConvert := 8102;
        RETURN;
    8111:
        FuUnicodeCodepointCaseConvert := 8103;
        RETURN;
    8112:
        FuUnicodeCodepointCaseConvert := 8120;
        RETURN;
    8113:
        FuUnicodeCodepointCaseConvert := 8121;
        RETURN;
    8115:
        FuUnicodeCodepointCaseConvert := 8124;
        RETURN;
    8120:
        FuUnicodeCodepointCaseConvert := 8112;
        RETURN;
    8121:
        FuUnicodeCodepointCaseConvert := 8113;
        RETURN;
    8122:
        FuUnicodeCodepointCaseConvert := 8048;
        RETURN;
    8123:
        FuUnicodeCodepointCaseConvert := 8049;
        RETURN;
    8124:
        FuUnicodeCodepointCaseConvert := 8115;
        RETURN;
    8126:
        FuUnicodeCodepointCaseConvert := 921;
        RETURN;
    8131:
        FuUnicodeCodepointCaseConvert := 8140;
        RETURN;
    8136:
        FuUnicodeCodepointCaseConvert := 8050;
        RETURN;
    8137:
        FuUnicodeCodepointCaseConvert := 8051;
        RETURN;
    8138:
        FuUnicodeCodepointCaseConvert := 8052;
        RETURN;
    8139:
        FuUnicodeCodepointCaseConvert := 8053;
        RETURN;
    8140:
        FuUnicodeCodepointCaseConvert := 8131;
        RETURN;
    8144:
        FuUnicodeCodepointCaseConvert := 8152;
        RETURN;
    8145:
        FuUnicodeCodepointCaseConvert := 8153;
        RETURN;
    8152:
        FuUnicodeCodepointCaseConvert := 8144;
        RETURN;
    8153:
        FuUnicodeCodepointCaseConvert := 8145;
        RETURN;
    8154:
        FuUnicodeCodepointCaseConvert := 8054;
        RETURN;
    8155:
        FuUnicodeCodepointCaseConvert := 8055;
        RETURN;
    8160:
        FuUnicodeCodepointCaseConvert := 8168;
        RETURN;
    8161:
        FuUnicodeCodepointCaseConvert := 8169;
        RETURN;
    8165:
        FuUnicodeCodepointCaseConvert := 8172;
        RETURN;
    8168:
        FuUnicodeCodepointCaseConvert := 8160;
        RETURN;
    8169:
        FuUnicodeCodepointCaseConvert := 8161;
        RETURN;
    8170:
        FuUnicodeCodepointCaseConvert := 8058;
        RETURN;
    8171:
        FuUnicodeCodepointCaseConvert := 8059;
        RETURN;
    8172:
        FuUnicodeCodepointCaseConvert := 8165;
        RETURN;
    8179:
        FuUnicodeCodepointCaseConvert := 8188;
        RETURN;
    8184:
        FuUnicodeCodepointCaseConvert := 8056;
        RETURN;
    8185:
        FuUnicodeCodepointCaseConvert := 8057;
        RETURN;
    8186:
        FuUnicodeCodepointCaseConvert := 8060;
        RETURN;
    8187:
        FuUnicodeCodepointCaseConvert := 8061;
        RETURN;
    8188:
        FuUnicodeCodepointCaseConvert := 8179;
        RETURN;
    8486:
        FuUnicodeCodepointCaseConvert := 969;
        RETURN;
    8490:
        FuUnicodeCodepointCaseConvert := 107;
        RETURN;
    8491:
        FuUnicodeCodepointCaseConvert := 229;
        RETURN;
    8498:
        FuUnicodeCodepointCaseConvert := 8526;
        RETURN;
    8526:
        FuUnicodeCodepointCaseConvert := 8498;
        RETURN;
    8544:
        FuUnicodeCodepointCaseConvert := 8560;
        RETURN;
    8545:
        FuUnicodeCodepointCaseConvert := 8561;
        RETURN;
    8546:
        FuUnicodeCodepointCaseConvert := 8562;
        RETURN;
    8547:
        FuUnicodeCodepointCaseConvert := 8563;
        RETURN;
    8548:
        FuUnicodeCodepointCaseConvert := 8564;
        RETURN;
    8549:
        FuUnicodeCodepointCaseConvert := 8565;
        RETURN;
    8550:
        FuUnicodeCodepointCaseConvert := 8566;
        RETURN;
    8551:
        FuUnicodeCodepointCaseConvert := 8567;
        RETURN;
    8552:
        FuUnicodeCodepointCaseConvert := 8568;
        RETURN;
    8553:
        FuUnicodeCodepointCaseConvert := 8569;
        RETURN;
    8554:
        FuUnicodeCodepointCaseConvert := 8570;
        RETURN;
    8555:
        FuUnicodeCodepointCaseConvert := 8571;
        RETURN;
    8556:
        FuUnicodeCodepointCaseConvert := 8572;
        RETURN;
    8557:
        FuUnicodeCodepointCaseConvert := 8573;
        RETURN;
    8558:
        FuUnicodeCodepointCaseConvert := 8574;
        RETURN;
    8559:
        FuUnicodeCodepointCaseConvert := 8575;
        RETURN;
    8560:
        FuUnicodeCodepointCaseConvert := 8544;
        RETURN;
    8561:
        FuUnicodeCodepointCaseConvert := 8545;
        RETURN;
    8562:
        FuUnicodeCodepointCaseConvert := 8546;
        RETURN;
    8563:
        FuUnicodeCodepointCaseConvert := 8547;
        RETURN;
    8564:
        FuUnicodeCodepointCaseConvert := 8548;
        RETURN;
    8565:
        FuUnicodeCodepointCaseConvert := 8549;
        RETURN;
    8566:
        FuUnicodeCodepointCaseConvert := 8550;
        RETURN;
    8567:
        FuUnicodeCodepointCaseConvert := 8551;
        RETURN;
    8568:
        FuUnicodeCodepointCaseConvert := 8552;
        RETURN;
    8569:
        FuUnicodeCodepointCaseConvert := 8553;
        RETURN;
    8570:
        FuUnicodeCodepointCaseConvert := 8554;
        RETURN;
    8571:
        FuUnicodeCodepointCaseConvert := 8555;
        RETURN;
    8572:
        FuUnicodeCodepointCaseConvert := 8556;
        RETURN;
    8573:
        FuUnicodeCodepointCaseConvert := 8557;
        RETURN;
    8574:
        FuUnicodeCodepointCaseConvert := 8558;
        RETURN;
    8575:
        FuUnicodeCodepointCaseConvert := 8559;
        RETURN;
    8579:
        FuUnicodeCodepointCaseConvert := 8580;
        RETURN;
    8580:
        FuUnicodeCodepointCaseConvert := 8579;
        RETURN;
    9398:
        FuUnicodeCodepointCaseConvert := 9424;
        RETURN;
    9399:
        FuUnicodeCodepointCaseConvert := 9425;
        RETURN;
    9400:
        FuUnicodeCodepointCaseConvert := 9426;
        RETURN;
    9401:
        FuUnicodeCodepointCaseConvert := 9427;
        RETURN;
    9402:
        FuUnicodeCodepointCaseConvert := 9428;
        RETURN;
    9403:
        FuUnicodeCodepointCaseConvert := 9429;
        RETURN;
    9404:
        FuUnicodeCodepointCaseConvert := 9430;
        RETURN;
    9405:
        FuUnicodeCodepointCaseConvert := 9431;
        RETURN;
    9406:
        FuUnicodeCodepointCaseConvert := 9432;
        RETURN;
    9407:
        FuUnicodeCodepointCaseConvert := 9433;
        RETURN;
    9408:
        FuUnicodeCodepointCaseConvert := 9434;
        RETURN;
    9409:
        FuUnicodeCodepointCaseConvert := 9435;
        RETURN;
    9410:
        FuUnicodeCodepointCaseConvert := 9436;
        RETURN;
    9411:
        FuUnicodeCodepointCaseConvert := 9437;
        RETURN;
    9412:
        FuUnicodeCodepointCaseConvert := 9438;
        RETURN;
    9413:
        FuUnicodeCodepointCaseConvert := 9439;
        RETURN;
    9414:
        FuUnicodeCodepointCaseConvert := 9440;
        RETURN;
    9415:
        FuUnicodeCodepointCaseConvert := 9441;
        RETURN;
    9416:
        FuUnicodeCodepointCaseConvert := 9442;
        RETURN;
    9417:
        FuUnicodeCodepointCaseConvert := 9443;
        RETURN;
    9418:
        FuUnicodeCodepointCaseConvert := 9444;
        RETURN;
    9419:
        FuUnicodeCodepointCaseConvert := 9445;
        RETURN;
    9420:
        FuUnicodeCodepointCaseConvert := 9446;
        RETURN;
    9421:
        FuUnicodeCodepointCaseConvert := 9447;
        RETURN;
    9422:
        FuUnicodeCodepointCaseConvert := 9448;
        RETURN;
    9423:
        FuUnicodeCodepointCaseConvert := 9449;
        RETURN;
    9424:
        FuUnicodeCodepointCaseConvert := 9398;
        RETURN;
    9425:
        FuUnicodeCodepointCaseConvert := 9399;
        RETURN;
    9426:
        FuUnicodeCodepointCaseConvert := 9400;
        RETURN;
    9427:
        FuUnicodeCodepointCaseConvert := 9401;
        RETURN;
    9428:
        FuUnicodeCodepointCaseConvert := 9402;
        RETURN;
    9429:
        FuUnicodeCodepointCaseConvert := 9403;
        RETURN;
    9430:
        FuUnicodeCodepointCaseConvert := 9404;
        RETURN;
    9431:
        FuUnicodeCodepointCaseConvert := 9405;
        RETURN;
    9432:
        FuUnicodeCodepointCaseConvert := 9406;
        RETURN;
    9433:
        FuUnicodeCodepointCaseConvert := 9407;
        RETURN;
    9434:
        FuUnicodeCodepointCaseConvert := 9408;
        RETURN;
    9435:
        FuUnicodeCodepointCaseConvert := 9409;
        RETURN;
    9436:
        FuUnicodeCodepointCaseConvert := 9410;
        RETURN;
    9437:
        FuUnicodeCodepointCaseConvert := 9411;
        RETURN;
    9438:
        FuUnicodeCodepointCaseConvert := 9412;
        RETURN;
    9439:
        FuUnicodeCodepointCaseConvert := 9413;
        RETURN;
    9440:
        FuUnicodeCodepointCaseConvert := 9414;
        RETURN;
    9441:
        FuUnicodeCodepointCaseConvert := 9415;
        RETURN;
    9442:
        FuUnicodeCodepointCaseConvert := 9416;
        RETURN;
    9443:
        FuUnicodeCodepointCaseConvert := 9417;
        RETURN;
    9444:
        FuUnicodeCodepointCaseConvert := 9418;
        RETURN;
    9445:
        FuUnicodeCodepointCaseConvert := 9419;
        RETURN;
    9446:
        FuUnicodeCodepointCaseConvert := 9420;
        RETURN;
    9447:
        FuUnicodeCodepointCaseConvert := 9421;
        RETURN;
    9448:
        FuUnicodeCodepointCaseConvert := 9422;
        RETURN;
    9449:
        FuUnicodeCodepointCaseConvert := 9423;
        RETURN;
    11264:
        FuUnicodeCodepointCaseConvert := 11312;
        RETURN;
    11265:
        FuUnicodeCodepointCaseConvert := 11313;
        RETURN;
    11266:
        FuUnicodeCodepointCaseConvert := 11314;
        RETURN;
    11267:
        FuUnicodeCodepointCaseConvert := 11315;
        RETURN;
    11268:
        FuUnicodeCodepointCaseConvert := 11316;
        RETURN;
    11269:
        FuUnicodeCodepointCaseConvert := 11317;
        RETURN;
    11270:
        FuUnicodeCodepointCaseConvert := 11318;
        RETURN;
    11271:
        FuUnicodeCodepointCaseConvert := 11319;
        RETURN;
    11272:
        FuUnicodeCodepointCaseConvert := 11320;
        RETURN;
    11273:
        FuUnicodeCodepointCaseConvert := 11321;
        RETURN;
    11274:
        FuUnicodeCodepointCaseConvert := 11322;
        RETURN;
    11275:
        FuUnicodeCodepointCaseConvert := 11323;
        RETURN;
    11276:
        FuUnicodeCodepointCaseConvert := 11324;
        RETURN;
    11277:
        FuUnicodeCodepointCaseConvert := 11325;
        RETURN;
    11278:
        FuUnicodeCodepointCaseConvert := 11326;
        RETURN;
    11279:
        FuUnicodeCodepointCaseConvert := 11327;
        RETURN;
    11280:
        FuUnicodeCodepointCaseConvert := 11328;
        RETURN;
    11281:
        FuUnicodeCodepointCaseConvert := 11329;
        RETURN;
    11282:
        FuUnicodeCodepointCaseConvert := 11330;
        RETURN;
    11283:
        FuUnicodeCodepointCaseConvert := 11331;
        RETURN;
    11284:
        FuUnicodeCodepointCaseConvert := 11332;
        RETURN;
    11285:
        FuUnicodeCodepointCaseConvert := 11333;
        RETURN;
    11286:
        FuUnicodeCodepointCaseConvert := 11334;
        RETURN;
    11287:
        FuUnicodeCodepointCaseConvert := 11335;
        RETURN;
    11288:
        FuUnicodeCodepointCaseConvert := 11336;
        RETURN;
    11289:
        FuUnicodeCodepointCaseConvert := 11337;
        RETURN;
    11290:
        FuUnicodeCodepointCaseConvert := 11338;
        RETURN;
    11291:
        FuUnicodeCodepointCaseConvert := 11339;
        RETURN;
    11292:
        FuUnicodeCodepointCaseConvert := 11340;
        RETURN;
    11293:
        FuUnicodeCodepointCaseConvert := 11341;
        RETURN;
    11294:
        FuUnicodeCodepointCaseConvert := 11342;
        RETURN;
    11295:
        FuUnicodeCodepointCaseConvert := 11343;
        RETURN;
    11296:
        FuUnicodeCodepointCaseConvert := 11344;
        RETURN;
    11297:
        FuUnicodeCodepointCaseConvert := 11345;
        RETURN;
    11298:
        FuUnicodeCodepointCaseConvert := 11346;
        RETURN;
    11299:
        FuUnicodeCodepointCaseConvert := 11347;
        RETURN;
    11300:
        FuUnicodeCodepointCaseConvert := 11348;
        RETURN;
    11301:
        FuUnicodeCodepointCaseConvert := 11349;
        RETURN;
    11302:
        FuUnicodeCodepointCaseConvert := 11350;
        RETURN;
    11303:
        FuUnicodeCodepointCaseConvert := 11351;
        RETURN;
    11304:
        FuUnicodeCodepointCaseConvert := 11352;
        RETURN;
    11305:
        FuUnicodeCodepointCaseConvert := 11353;
        RETURN;
    11306:
        FuUnicodeCodepointCaseConvert := 11354;
        RETURN;
    11307:
        FuUnicodeCodepointCaseConvert := 11355;
        RETURN;
    11308:
        FuUnicodeCodepointCaseConvert := 11356;
        RETURN;
    11309:
        FuUnicodeCodepointCaseConvert := 11357;
        RETURN;
    11310:
        FuUnicodeCodepointCaseConvert := 11358;
        RETURN;
    11311:
        FuUnicodeCodepointCaseConvert := 11359;
        RETURN;
    11312:
        FuUnicodeCodepointCaseConvert := 11264;
        RETURN;
    11313:
        FuUnicodeCodepointCaseConvert := 11265;
        RETURN;
    11314:
        FuUnicodeCodepointCaseConvert := 11266;
        RETURN;
    11315:
        FuUnicodeCodepointCaseConvert := 11267;
        RETURN;
    11316:
        FuUnicodeCodepointCaseConvert := 11268;
        RETURN;
    11317:
        FuUnicodeCodepointCaseConvert := 11269;
        RETURN;
    11318:
        FuUnicodeCodepointCaseConvert := 11270;
        RETURN;
    11319:
        FuUnicodeCodepointCaseConvert := 11271;
        RETURN;
    11320:
        FuUnicodeCodepointCaseConvert := 11272;
        RETURN;
    11321:
        FuUnicodeCodepointCaseConvert := 11273;
        RETURN;
    11322:
        FuUnicodeCodepointCaseConvert := 11274;
        RETURN;
    11323:
        FuUnicodeCodepointCaseConvert := 11275;
        RETURN;
    11324:
        FuUnicodeCodepointCaseConvert := 11276;
        RETURN;
    11325:
        FuUnicodeCodepointCaseConvert := 11277;
        RETURN;
    11326:
        FuUnicodeCodepointCaseConvert := 11278;
        RETURN;
    11327:
        FuUnicodeCodepointCaseConvert := 11279;
        RETURN;
    11328:
        FuUnicodeCodepointCaseConvert := 11280;
        RETURN;
    11329:
        FuUnicodeCodepointCaseConvert := 11281;
        RETURN;
    11330:
        FuUnicodeCodepointCaseConvert := 11282;
        RETURN;
    11331:
        FuUnicodeCodepointCaseConvert := 11283;
        RETURN;
    11332:
        FuUnicodeCodepointCaseConvert := 11284;
        RETURN;
    11333:
        FuUnicodeCodepointCaseConvert := 11285;
        RETURN;
    11334:
        FuUnicodeCodepointCaseConvert := 11286;
        RETURN;
    11335:
        FuUnicodeCodepointCaseConvert := 11287;
        RETURN;
    11336:
        FuUnicodeCodepointCaseConvert := 11288;
        RETURN;
    11337:
        FuUnicodeCodepointCaseConvert := 11289;
        RETURN;
    11338:
        FuUnicodeCodepointCaseConvert := 11290;
        RETURN;
    11339:
        FuUnicodeCodepointCaseConvert := 11291;
        RETURN;
    11340:
        FuUnicodeCodepointCaseConvert := 11292;
        RETURN;
    11341:
        FuUnicodeCodepointCaseConvert := 11293;
        RETURN;
    11342:
        FuUnicodeCodepointCaseConvert := 11294;
        RETURN;
    11343:
        FuUnicodeCodepointCaseConvert := 11295;
        RETURN;
    11344:
        FuUnicodeCodepointCaseConvert := 11296;
        RETURN;
    11345:
        FuUnicodeCodepointCaseConvert := 11297;
        RETURN;
    11346:
        FuUnicodeCodepointCaseConvert := 11298;
        RETURN;
    11347:
        FuUnicodeCodepointCaseConvert := 11299;
        RETURN;
    11348:
        FuUnicodeCodepointCaseConvert := 11300;
        RETURN;
    11349:
        FuUnicodeCodepointCaseConvert := 11301;
        RETURN;
    11350:
        FuUnicodeCodepointCaseConvert := 11302;
        RETURN;
    11351:
        FuUnicodeCodepointCaseConvert := 11303;
        RETURN;
    11352:
        FuUnicodeCodepointCaseConvert := 11304;
        RETURN;
    11353:
        FuUnicodeCodepointCaseConvert := 11305;
        RETURN;
    11354:
        FuUnicodeCodepointCaseConvert := 11306;
        RETURN;
    11355:
        FuUnicodeCodepointCaseConvert := 11307;
        RETURN;
    11356:
        FuUnicodeCodepointCaseConvert := 11308;
        RETURN;
    11357:
        FuUnicodeCodepointCaseConvert := 11309;
        RETURN;
    11358:
        FuUnicodeCodepointCaseConvert := 11310;
        RETURN;
    11359:
        FuUnicodeCodepointCaseConvert := 11311;
        RETURN;
    11360:
        FuUnicodeCodepointCaseConvert := 11361;
        RETURN;
    11361:
        FuUnicodeCodepointCaseConvert := 11360;
        RETURN;
    11362:
        FuUnicodeCodepointCaseConvert := 619;
        RETURN;
    11363:
        FuUnicodeCodepointCaseConvert := 7549;
        RETURN;
    11364:
        FuUnicodeCodepointCaseConvert := 637;
        RETURN;
    11365:
        FuUnicodeCodepointCaseConvert := 570;
        RETURN;
    11366:
        FuUnicodeCodepointCaseConvert := 574;
        RETURN;
    11367:
        FuUnicodeCodepointCaseConvert := 11368;
        RETURN;
    11368:
        FuUnicodeCodepointCaseConvert := 11367;
        RETURN;
    11369:
        FuUnicodeCodepointCaseConvert := 11370;
        RETURN;
    11370:
        FuUnicodeCodepointCaseConvert := 11369;
        RETURN;
    11371:
        FuUnicodeCodepointCaseConvert := 11372;
        RETURN;
    11372:
        FuUnicodeCodepointCaseConvert := 11371;
        RETURN;
    11373:
        FuUnicodeCodepointCaseConvert := 593;
        RETURN;
    11374:
        FuUnicodeCodepointCaseConvert := 625;
        RETURN;
    11375:
        FuUnicodeCodepointCaseConvert := 592;
        RETURN;
    11376:
        FuUnicodeCodepointCaseConvert := 594;
        RETURN;
    11378:
        FuUnicodeCodepointCaseConvert := 11379;
        RETURN;
    11379:
        FuUnicodeCodepointCaseConvert := 11378;
        RETURN;
    11381:
        FuUnicodeCodepointCaseConvert := 11382;
        RETURN;
    11382:
        FuUnicodeCodepointCaseConvert := 11381;
        RETURN;
    11390:
        FuUnicodeCodepointCaseConvert := 575;
        RETURN;
    11391:
        FuUnicodeCodepointCaseConvert := 576;
        RETURN;
    11392:
        FuUnicodeCodepointCaseConvert := 11393;
        RETURN;
    11393:
        FuUnicodeCodepointCaseConvert := 11392;
        RETURN;
    11394:
        FuUnicodeCodepointCaseConvert := 11395;
        RETURN;
    11395:
        FuUnicodeCodepointCaseConvert := 11394;
        RETURN;
    11396:
        FuUnicodeCodepointCaseConvert := 11397;
        RETURN;
    11397:
        FuUnicodeCodepointCaseConvert := 11396;
        RETURN;
    11398:
        FuUnicodeCodepointCaseConvert := 11399;
        RETURN;
    11399:
        FuUnicodeCodepointCaseConvert := 11398;
        RETURN;
    11400:
        FuUnicodeCodepointCaseConvert := 11401;
        RETURN;
    11401:
        FuUnicodeCodepointCaseConvert := 11400;
        RETURN;
    11402:
        FuUnicodeCodepointCaseConvert := 11403;
        RETURN;
    11403:
        FuUnicodeCodepointCaseConvert := 11402;
        RETURN;
    11404:
        FuUnicodeCodepointCaseConvert := 11405;
        RETURN;
    11405:
        FuUnicodeCodepointCaseConvert := 11404;
        RETURN;
    11406:
        FuUnicodeCodepointCaseConvert := 11407;
        RETURN;
    11407:
        FuUnicodeCodepointCaseConvert := 11406;
        RETURN;
    11408:
        FuUnicodeCodepointCaseConvert := 11409;
        RETURN;
    11409:
        FuUnicodeCodepointCaseConvert := 11408;
        RETURN;
    11410:
        FuUnicodeCodepointCaseConvert := 11411;
        RETURN;
    11411:
        FuUnicodeCodepointCaseConvert := 11410;
        RETURN;
    11412:
        FuUnicodeCodepointCaseConvert := 11413;
        RETURN;
    11413:
        FuUnicodeCodepointCaseConvert := 11412;
        RETURN;
    11414:
        FuUnicodeCodepointCaseConvert := 11415;
        RETURN;
    11415:
        FuUnicodeCodepointCaseConvert := 11414;
        RETURN;
    11416:
        FuUnicodeCodepointCaseConvert := 11417;
        RETURN;
    11417:
        FuUnicodeCodepointCaseConvert := 11416;
        RETURN;
    11418:
        FuUnicodeCodepointCaseConvert := 11419;
        RETURN;
    11419:
        FuUnicodeCodepointCaseConvert := 11418;
        RETURN;
    11420:
        FuUnicodeCodepointCaseConvert := 11421;
        RETURN;
    11421:
        FuUnicodeCodepointCaseConvert := 11420;
        RETURN;
    11422:
        FuUnicodeCodepointCaseConvert := 11423;
        RETURN;
    11423:
        FuUnicodeCodepointCaseConvert := 11422;
        RETURN;
    11424:
        FuUnicodeCodepointCaseConvert := 11425;
        RETURN;
    11425:
        FuUnicodeCodepointCaseConvert := 11424;
        RETURN;
    11426:
        FuUnicodeCodepointCaseConvert := 11427;
        RETURN;
    11427:
        FuUnicodeCodepointCaseConvert := 11426;
        RETURN;
    11428:
        FuUnicodeCodepointCaseConvert := 11429;
        RETURN;
    11429:
        FuUnicodeCodepointCaseConvert := 11428;
        RETURN;
    11430:
        FuUnicodeCodepointCaseConvert := 11431;
        RETURN;
    11431:
        FuUnicodeCodepointCaseConvert := 11430;
        RETURN;
    11432:
        FuUnicodeCodepointCaseConvert := 11433;
        RETURN;
    11433:
        FuUnicodeCodepointCaseConvert := 11432;
        RETURN;
    11434:
        FuUnicodeCodepointCaseConvert := 11435;
        RETURN;
    11435:
        FuUnicodeCodepointCaseConvert := 11434;
        RETURN;
    11436:
        FuUnicodeCodepointCaseConvert := 11437;
        RETURN;
    11437:
        FuUnicodeCodepointCaseConvert := 11436;
        RETURN;
    11438:
        FuUnicodeCodepointCaseConvert := 11439;
        RETURN;
    11439:
        FuUnicodeCodepointCaseConvert := 11438;
        RETURN;
    11440:
        FuUnicodeCodepointCaseConvert := 11441;
        RETURN;
    11441:
        FuUnicodeCodepointCaseConvert := 11440;
        RETURN;
    11442:
        FuUnicodeCodepointCaseConvert := 11443;
        RETURN;
    11443:
        FuUnicodeCodepointCaseConvert := 11442;
        RETURN;
    11444:
        FuUnicodeCodepointCaseConvert := 11445;
        RETURN;
    11445:
        FuUnicodeCodepointCaseConvert := 11444;
        RETURN;
    11446:
        FuUnicodeCodepointCaseConvert := 11447;
        RETURN;
    11447:
        FuUnicodeCodepointCaseConvert := 11446;
        RETURN;
    11448:
        FuUnicodeCodepointCaseConvert := 11449;
        RETURN;
    11449:
        FuUnicodeCodepointCaseConvert := 11448;
        RETURN;
    11450:
        FuUnicodeCodepointCaseConvert := 11451;
        RETURN;
    11451:
        FuUnicodeCodepointCaseConvert := 11450;
        RETURN;
    11452:
        FuUnicodeCodepointCaseConvert := 11453;
        RETURN;
    11453:
        FuUnicodeCodepointCaseConvert := 11452;
        RETURN;
    11454:
        FuUnicodeCodepointCaseConvert := 11455;
        RETURN;
    11455:
        FuUnicodeCodepointCaseConvert := 11454;
        RETURN;
    11456:
        FuUnicodeCodepointCaseConvert := 11457;
        RETURN;
    11457:
        FuUnicodeCodepointCaseConvert := 11456;
        RETURN;
    11458:
        FuUnicodeCodepointCaseConvert := 11459;
        RETURN;
    11459:
        FuUnicodeCodepointCaseConvert := 11458;
        RETURN;
    11460:
        FuUnicodeCodepointCaseConvert := 11461;
        RETURN;
    11461:
        FuUnicodeCodepointCaseConvert := 11460;
        RETURN;
    11462:
        FuUnicodeCodepointCaseConvert := 11463;
        RETURN;
    11463:
        FuUnicodeCodepointCaseConvert := 11462;
        RETURN;
    11464:
        FuUnicodeCodepointCaseConvert := 11465;
        RETURN;
    11465:
        FuUnicodeCodepointCaseConvert := 11464;
        RETURN;
    11466:
        FuUnicodeCodepointCaseConvert := 11467;
        RETURN;
    11467:
        FuUnicodeCodepointCaseConvert := 11466;
        RETURN;
    11468:
        FuUnicodeCodepointCaseConvert := 11469;
        RETURN;
    11469:
        FuUnicodeCodepointCaseConvert := 11468;
        RETURN;
    11470:
        FuUnicodeCodepointCaseConvert := 11471;
        RETURN;
    11471:
        FuUnicodeCodepointCaseConvert := 11470;
        RETURN;
    11472:
        FuUnicodeCodepointCaseConvert := 11473;
        RETURN;
    11473:
        FuUnicodeCodepointCaseConvert := 11472;
        RETURN;
    11474:
        FuUnicodeCodepointCaseConvert := 11475;
        RETURN;
    11475:
        FuUnicodeCodepointCaseConvert := 11474;
        RETURN;
    11476:
        FuUnicodeCodepointCaseConvert := 11477;
        RETURN;
    11477:
        FuUnicodeCodepointCaseConvert := 11476;
        RETURN;
    11478:
        FuUnicodeCodepointCaseConvert := 11479;
        RETURN;
    11479:
        FuUnicodeCodepointCaseConvert := 11478;
        RETURN;
    11480:
        FuUnicodeCodepointCaseConvert := 11481;
        RETURN;
    11481:
        FuUnicodeCodepointCaseConvert := 11480;
        RETURN;
    11482:
        FuUnicodeCodepointCaseConvert := 11483;
        RETURN;
    11483:
        FuUnicodeCodepointCaseConvert := 11482;
        RETURN;
    11484:
        FuUnicodeCodepointCaseConvert := 11485;
        RETURN;
    11485:
        FuUnicodeCodepointCaseConvert := 11484;
        RETURN;
    11486:
        FuUnicodeCodepointCaseConvert := 11487;
        RETURN;
    11487:
        FuUnicodeCodepointCaseConvert := 11486;
        RETURN;
    11488:
        FuUnicodeCodepointCaseConvert := 11489;
        RETURN;
    11489:
        FuUnicodeCodepointCaseConvert := 11488;
        RETURN;
    11490:
        FuUnicodeCodepointCaseConvert := 11491;
        RETURN;
    11491:
        FuUnicodeCodepointCaseConvert := 11490;
        RETURN;
    11499:
        FuUnicodeCodepointCaseConvert := 11500;
        RETURN;
    11500:
        FuUnicodeCodepointCaseConvert := 11499;
        RETURN;
    11501:
        FuUnicodeCodepointCaseConvert := 11502;
        RETURN;
    11502:
        FuUnicodeCodepointCaseConvert := 11501;
        RETURN;
    11506:
        FuUnicodeCodepointCaseConvert := 11507;
        RETURN;
    11507:
        FuUnicodeCodepointCaseConvert := 11506;
        RETURN;
    11520:
        FuUnicodeCodepointCaseConvert := 4256;
        RETURN;
    11521:
        FuUnicodeCodepointCaseConvert := 4257;
        RETURN;
    11522:
        FuUnicodeCodepointCaseConvert := 4258;
        RETURN;
    11523:
        FuUnicodeCodepointCaseConvert := 4259;
        RETURN;
    11524:
        FuUnicodeCodepointCaseConvert := 4260;
        RETURN;
    11525:
        FuUnicodeCodepointCaseConvert := 4261;
        RETURN;
    11526:
        FuUnicodeCodepointCaseConvert := 4262;
        RETURN;
    11527:
        FuUnicodeCodepointCaseConvert := 4263;
        RETURN;
    11528:
        FuUnicodeCodepointCaseConvert := 4264;
        RETURN;
    11529:
        FuUnicodeCodepointCaseConvert := 4265;
        RETURN;
    11530:
        FuUnicodeCodepointCaseConvert := 4266;
        RETURN;
    11531:
        FuUnicodeCodepointCaseConvert := 4267;
        RETURN;
    11532:
        FuUnicodeCodepointCaseConvert := 4268;
        RETURN;
    11533:
        FuUnicodeCodepointCaseConvert := 4269;
        RETURN;
    11534:
        FuUnicodeCodepointCaseConvert := 4270;
        RETURN;
    11535:
        FuUnicodeCodepointCaseConvert := 4271;
        RETURN;
    11536:
        FuUnicodeCodepointCaseConvert := 4272;
        RETURN;
    11537:
        FuUnicodeCodepointCaseConvert := 4273;
        RETURN;
    11538:
        FuUnicodeCodepointCaseConvert := 4274;
        RETURN;
    11539:
        FuUnicodeCodepointCaseConvert := 4275;
        RETURN;
    11540:
        FuUnicodeCodepointCaseConvert := 4276;
        RETURN;
    11541:
        FuUnicodeCodepointCaseConvert := 4277;
        RETURN;
    11542:
        FuUnicodeCodepointCaseConvert := 4278;
        RETURN;
    11543:
        FuUnicodeCodepointCaseConvert := 4279;
        RETURN;
    11544:
        FuUnicodeCodepointCaseConvert := 4280;
        RETURN;
    11545:
        FuUnicodeCodepointCaseConvert := 4281;
        RETURN;
    11546:
        FuUnicodeCodepointCaseConvert := 4282;
        RETURN;
    11547:
        FuUnicodeCodepointCaseConvert := 4283;
        RETURN;
    11548:
        FuUnicodeCodepointCaseConvert := 4284;
        RETURN;
    11549:
        FuUnicodeCodepointCaseConvert := 4285;
        RETURN;
    11550:
        FuUnicodeCodepointCaseConvert := 4286;
        RETURN;
    11551:
        FuUnicodeCodepointCaseConvert := 4287;
        RETURN;
    11552:
        FuUnicodeCodepointCaseConvert := 4288;
        RETURN;
    11553:
        FuUnicodeCodepointCaseConvert := 4289;
        RETURN;
    11554:
        FuUnicodeCodepointCaseConvert := 4290;
        RETURN;
    11555:
        FuUnicodeCodepointCaseConvert := 4291;
        RETURN;
    11556:
        FuUnicodeCodepointCaseConvert := 4292;
        RETURN;
    11557:
        FuUnicodeCodepointCaseConvert := 4293;
        RETURN;
    11559:
        FuUnicodeCodepointCaseConvert := 4295;
        RETURN;
    11565:
        FuUnicodeCodepointCaseConvert := 4301;
        RETURN;
    42560:
        FuUnicodeCodepointCaseConvert := 42561;
        RETURN;
    42561:
        FuUnicodeCodepointCaseConvert := 42560;
        RETURN;
    42562:
        FuUnicodeCodepointCaseConvert := 42563;
        RETURN;
    42563:
        FuUnicodeCodepointCaseConvert := 42562;
        RETURN;
    42564:
        FuUnicodeCodepointCaseConvert := 42565;
        RETURN;
    42565:
        FuUnicodeCodepointCaseConvert := 42564;
        RETURN;
    42566:
        FuUnicodeCodepointCaseConvert := 42567;
        RETURN;
    42567:
        FuUnicodeCodepointCaseConvert := 42566;
        RETURN;
    42568:
        FuUnicodeCodepointCaseConvert := 42569;
        RETURN;
    42569:
        FuUnicodeCodepointCaseConvert := 42568;
        RETURN;
    42570:
        FuUnicodeCodepointCaseConvert := 42571;
        RETURN;
    42571:
        FuUnicodeCodepointCaseConvert := 42570;
        RETURN;
    42572:
        FuUnicodeCodepointCaseConvert := 42573;
        RETURN;
    42573:
        FuUnicodeCodepointCaseConvert := 42572;
        RETURN;
    42574:
        FuUnicodeCodepointCaseConvert := 42575;
        RETURN;
    42575:
        FuUnicodeCodepointCaseConvert := 42574;
        RETURN;
    42576:
        FuUnicodeCodepointCaseConvert := 42577;
        RETURN;
    42577:
        FuUnicodeCodepointCaseConvert := 42576;
        RETURN;
    42578:
        FuUnicodeCodepointCaseConvert := 42579;
        RETURN;
    42579:
        FuUnicodeCodepointCaseConvert := 42578;
        RETURN;
    42580:
        FuUnicodeCodepointCaseConvert := 42581;
        RETURN;
    42581:
        FuUnicodeCodepointCaseConvert := 42580;
        RETURN;
    42582:
        FuUnicodeCodepointCaseConvert := 42583;
        RETURN;
    42583:
        FuUnicodeCodepointCaseConvert := 42582;
        RETURN;
    42584:
        FuUnicodeCodepointCaseConvert := 42585;
        RETURN;
    42585:
        FuUnicodeCodepointCaseConvert := 42584;
        RETURN;
    42586:
        FuUnicodeCodepointCaseConvert := 42587;
        RETURN;
    42587:
        FuUnicodeCodepointCaseConvert := 42586;
        RETURN;
    42588:
        FuUnicodeCodepointCaseConvert := 42589;
        RETURN;
    42589:
        FuUnicodeCodepointCaseConvert := 42588;
        RETURN;
    42590:
        FuUnicodeCodepointCaseConvert := 42591;
        RETURN;
    42591:
        FuUnicodeCodepointCaseConvert := 42590;
        RETURN;
    42592:
        FuUnicodeCodepointCaseConvert := 42593;
        RETURN;
    42593:
        FuUnicodeCodepointCaseConvert := 42592;
        RETURN;
    42594:
        FuUnicodeCodepointCaseConvert := 42595;
        RETURN;
    42595:
        FuUnicodeCodepointCaseConvert := 42594;
        RETURN;
    42596:
        FuUnicodeCodepointCaseConvert := 42597;
        RETURN;
    42597:
        FuUnicodeCodepointCaseConvert := 42596;
        RETURN;
    42598:
        FuUnicodeCodepointCaseConvert := 42599;
        RETURN;
    42599:
        FuUnicodeCodepointCaseConvert := 42598;
        RETURN;
    42600:
        FuUnicodeCodepointCaseConvert := 42601;
        RETURN;
    42601:
        FuUnicodeCodepointCaseConvert := 42600;
        RETURN;
    42602:
        FuUnicodeCodepointCaseConvert := 42603;
        RETURN;
    42603:
        FuUnicodeCodepointCaseConvert := 42602;
        RETURN;
    42604:
        FuUnicodeCodepointCaseConvert := 42605;
        RETURN;
    42605:
        FuUnicodeCodepointCaseConvert := 42604;
        RETURN;
    42624:
        FuUnicodeCodepointCaseConvert := 42625;
        RETURN;
    42625:
        FuUnicodeCodepointCaseConvert := 42624;
        RETURN;
    42626:
        FuUnicodeCodepointCaseConvert := 42627;
        RETURN;
    42627:
        FuUnicodeCodepointCaseConvert := 42626;
        RETURN;
    42628:
        FuUnicodeCodepointCaseConvert := 42629;
        RETURN;
    42629:
        FuUnicodeCodepointCaseConvert := 42628;
        RETURN;
    42630:
        FuUnicodeCodepointCaseConvert := 42631;
        RETURN;
    42631:
        FuUnicodeCodepointCaseConvert := 42630;
        RETURN;
    42632:
        FuUnicodeCodepointCaseConvert := 42633;
        RETURN;
    42633:
        FuUnicodeCodepointCaseConvert := 42632;
        RETURN;
    42634:
        FuUnicodeCodepointCaseConvert := 42635;
        RETURN;
    42635:
        FuUnicodeCodepointCaseConvert := 42634;
        RETURN;
    42636:
        FuUnicodeCodepointCaseConvert := 42637;
        RETURN;
    42637:
        FuUnicodeCodepointCaseConvert := 42636;
        RETURN;
    42638:
        FuUnicodeCodepointCaseConvert := 42639;
        RETURN;
    42639:
        FuUnicodeCodepointCaseConvert := 42638;
        RETURN;
    42640:
        FuUnicodeCodepointCaseConvert := 42641;
        RETURN;
    42641:
        FuUnicodeCodepointCaseConvert := 42640;
        RETURN;
    42642:
        FuUnicodeCodepointCaseConvert := 42643;
        RETURN;
    42643:
        FuUnicodeCodepointCaseConvert := 42642;
        RETURN;
    42644:
        FuUnicodeCodepointCaseConvert := 42645;
        RETURN;
    42645:
        FuUnicodeCodepointCaseConvert := 42644;
        RETURN;
    42646:
        FuUnicodeCodepointCaseConvert := 42647;
        RETURN;
    42647:
        FuUnicodeCodepointCaseConvert := 42646;
        RETURN;
    42648:
        FuUnicodeCodepointCaseConvert := 42649;
        RETURN;
    42649:
        FuUnicodeCodepointCaseConvert := 42648;
        RETURN;
    42650:
        FuUnicodeCodepointCaseConvert := 42651;
        RETURN;
    42651:
        FuUnicodeCodepointCaseConvert := 42650;
        RETURN;
    42786:
        FuUnicodeCodepointCaseConvert := 42787;
        RETURN;
    42787:
        FuUnicodeCodepointCaseConvert := 42786;
        RETURN;
    42788:
        FuUnicodeCodepointCaseConvert := 42789;
        RETURN;
    42789:
        FuUnicodeCodepointCaseConvert := 42788;
        RETURN;
    42790:
        FuUnicodeCodepointCaseConvert := 42791;
        RETURN;
    42791:
        FuUnicodeCodepointCaseConvert := 42790;
        RETURN;
    42792:
        FuUnicodeCodepointCaseConvert := 42793;
        RETURN;
    42793:
        FuUnicodeCodepointCaseConvert := 42792;
        RETURN;
    42794:
        FuUnicodeCodepointCaseConvert := 42795;
        RETURN;
    42795:
        FuUnicodeCodepointCaseConvert := 42794;
        RETURN;
    42796:
        FuUnicodeCodepointCaseConvert := 42797;
        RETURN;
    42797:
        FuUnicodeCodepointCaseConvert := 42796;
        RETURN;
    42798:
        FuUnicodeCodepointCaseConvert := 42799;
        RETURN;
    42799:
        FuUnicodeCodepointCaseConvert := 42798;
        RETURN;
    42802:
        FuUnicodeCodepointCaseConvert := 42803;
        RETURN;
    42803:
        FuUnicodeCodepointCaseConvert := 42802;
        RETURN;
    42804:
        FuUnicodeCodepointCaseConvert := 42805;
        RETURN;
    42805:
        FuUnicodeCodepointCaseConvert := 42804;
        RETURN;
    42806:
        FuUnicodeCodepointCaseConvert := 42807;
        RETURN;
    42807:
        FuUnicodeCodepointCaseConvert := 42806;
        RETURN;
    42808:
        FuUnicodeCodepointCaseConvert := 42809;
        RETURN;
    42809:
        FuUnicodeCodepointCaseConvert := 42808;
        RETURN;
    42810:
        FuUnicodeCodepointCaseConvert := 42811;
        RETURN;
    42811:
        FuUnicodeCodepointCaseConvert := 42810;
        RETURN;
    42812:
        FuUnicodeCodepointCaseConvert := 42813;
        RETURN;
    42813:
        FuUnicodeCodepointCaseConvert := 42812;
        RETURN;
    42814:
        FuUnicodeCodepointCaseConvert := 42815;
        RETURN;
    42815:
        FuUnicodeCodepointCaseConvert := 42814;
        RETURN;
    42816:
        FuUnicodeCodepointCaseConvert := 42817;
        RETURN;
    42817:
        FuUnicodeCodepointCaseConvert := 42816;
        RETURN;
    42818:
        FuUnicodeCodepointCaseConvert := 42819;
        RETURN;
    42819:
        FuUnicodeCodepointCaseConvert := 42818;
        RETURN;
    42820:
        FuUnicodeCodepointCaseConvert := 42821;
        RETURN;
    42821:
        FuUnicodeCodepointCaseConvert := 42820;
        RETURN;
    42822:
        FuUnicodeCodepointCaseConvert := 42823;
        RETURN;
    42823:
        FuUnicodeCodepointCaseConvert := 42822;
        RETURN;
    42824:
        FuUnicodeCodepointCaseConvert := 42825;
        RETURN;
    42825:
        FuUnicodeCodepointCaseConvert := 42824;
        RETURN;
    42826:
        FuUnicodeCodepointCaseConvert := 42827;
        RETURN;
    42827:
        FuUnicodeCodepointCaseConvert := 42826;
        RETURN;
    42828:
        FuUnicodeCodepointCaseConvert := 42829;
        RETURN;
    42829:
        FuUnicodeCodepointCaseConvert := 42828;
        RETURN;
    42830:
        FuUnicodeCodepointCaseConvert := 42831;
        RETURN;
    42831:
        FuUnicodeCodepointCaseConvert := 42830;
        RETURN;
    42832:
        FuUnicodeCodepointCaseConvert := 42833;
        RETURN;
    42833:
        FuUnicodeCodepointCaseConvert := 42832;
        RETURN;
    42834:
        FuUnicodeCodepointCaseConvert := 42835;
        RETURN;
    42835:
        FuUnicodeCodepointCaseConvert := 42834;
        RETURN;
    42836:
        FuUnicodeCodepointCaseConvert := 42837;
        RETURN;
    42837:
        FuUnicodeCodepointCaseConvert := 42836;
        RETURN;
    42838:
        FuUnicodeCodepointCaseConvert := 42839;
        RETURN;
    42839:
        FuUnicodeCodepointCaseConvert := 42838;
        RETURN;
    42840:
        FuUnicodeCodepointCaseConvert := 42841;
        RETURN;
    42841:
        FuUnicodeCodepointCaseConvert := 42840;
        RETURN;
    42842:
        FuUnicodeCodepointCaseConvert := 42843;
        RETURN;
    42843:
        FuUnicodeCodepointCaseConvert := 42842;
        RETURN;
    42844:
        FuUnicodeCodepointCaseConvert := 42845;
        RETURN;
    42845:
        FuUnicodeCodepointCaseConvert := 42844;
        RETURN;
    42846:
        FuUnicodeCodepointCaseConvert := 42847;
        RETURN;
    42847:
        FuUnicodeCodepointCaseConvert := 42846;
        RETURN;
    42848:
        FuUnicodeCodepointCaseConvert := 42849;
        RETURN;
    42849:
        FuUnicodeCodepointCaseConvert := 42848;
        RETURN;
    42850:
        FuUnicodeCodepointCaseConvert := 42851;
        RETURN;
    42851:
        FuUnicodeCodepointCaseConvert := 42850;
        RETURN;
    42852:
        FuUnicodeCodepointCaseConvert := 42853;
        RETURN;
    42853:
        FuUnicodeCodepointCaseConvert := 42852;
        RETURN;
    42854:
        FuUnicodeCodepointCaseConvert := 42855;
        RETURN;
    42855:
        FuUnicodeCodepointCaseConvert := 42854;
        RETURN;
    42856:
        FuUnicodeCodepointCaseConvert := 42857;
        RETURN;
    42857:
        FuUnicodeCodepointCaseConvert := 42856;
        RETURN;
    42858:
        FuUnicodeCodepointCaseConvert := 42859;
        RETURN;
    42859:
        FuUnicodeCodepointCaseConvert := 42858;
        RETURN;
    42860:
        FuUnicodeCodepointCaseConvert := 42861;
        RETURN;
    42861:
        FuUnicodeCodepointCaseConvert := 42860;
        RETURN;
    42862:
        FuUnicodeCodepointCaseConvert := 42863;
        RETURN;
    42863:
        FuUnicodeCodepointCaseConvert := 42862;
        RETURN;
    42873:
        FuUnicodeCodepointCaseConvert := 42874;
        RETURN;
    42874:
        FuUnicodeCodepointCaseConvert := 42873;
        RETURN;
    42875:
        FuUnicodeCodepointCaseConvert := 42876;
        RETURN;
    42876:
        FuUnicodeCodepointCaseConvert := 42875;
        RETURN;
    42877:
        FuUnicodeCodepointCaseConvert := 7545;
        RETURN;
    42878:
        FuUnicodeCodepointCaseConvert := 42879;
        RETURN;
    42879:
        FuUnicodeCodepointCaseConvert := 42878;
        RETURN;
    42880:
        FuUnicodeCodepointCaseConvert := 42881;
        RETURN;
    42881:
        FuUnicodeCodepointCaseConvert := 42880;
        RETURN;
    42882:
        FuUnicodeCodepointCaseConvert := 42883;
        RETURN;
    42883:
        FuUnicodeCodepointCaseConvert := 42882;
        RETURN;
    42884:
        FuUnicodeCodepointCaseConvert := 42885;
        RETURN;
    42885:
        FuUnicodeCodepointCaseConvert := 42884;
        RETURN;
    42886:
        FuUnicodeCodepointCaseConvert := 42887;
        RETURN;
    42887:
        FuUnicodeCodepointCaseConvert := 42886;
        RETURN;
    42891:
        FuUnicodeCodepointCaseConvert := 42892;
        RETURN;
    42892:
        FuUnicodeCodepointCaseConvert := 42891;
        RETURN;
    42893:
        FuUnicodeCodepointCaseConvert := 613;
        RETURN;
    42896:
        FuUnicodeCodepointCaseConvert := 42897;
        RETURN;
    42897:
        FuUnicodeCodepointCaseConvert := 42896;
        RETURN;
    42898:
        FuUnicodeCodepointCaseConvert := 42899;
        RETURN;
    42899:
        FuUnicodeCodepointCaseConvert := 42898;
        RETURN;
    42900:
        FuUnicodeCodepointCaseConvert := 42948;
        RETURN;
    42902:
        FuUnicodeCodepointCaseConvert := 42903;
        RETURN;
    42903:
        FuUnicodeCodepointCaseConvert := 42902;
        RETURN;
    42904:
        FuUnicodeCodepointCaseConvert := 42905;
        RETURN;
    42905:
        FuUnicodeCodepointCaseConvert := 42904;
        RETURN;
    42906:
        FuUnicodeCodepointCaseConvert := 42907;
        RETURN;
    42907:
        FuUnicodeCodepointCaseConvert := 42906;
        RETURN;
    42908:
        FuUnicodeCodepointCaseConvert := 42909;
        RETURN;
    42909:
        FuUnicodeCodepointCaseConvert := 42908;
        RETURN;
    42910:
        FuUnicodeCodepointCaseConvert := 42911;
        RETURN;
    42911:
        FuUnicodeCodepointCaseConvert := 42910;
        RETURN;
    42912:
        FuUnicodeCodepointCaseConvert := 42913;
        RETURN;
    42913:
        FuUnicodeCodepointCaseConvert := 42912;
        RETURN;
    42914:
        FuUnicodeCodepointCaseConvert := 42915;
        RETURN;
    42915:
        FuUnicodeCodepointCaseConvert := 42914;
        RETURN;
    42916:
        FuUnicodeCodepointCaseConvert := 42917;
        RETURN;
    42917:
        FuUnicodeCodepointCaseConvert := 42916;
        RETURN;
    42918:
        FuUnicodeCodepointCaseConvert := 42919;
        RETURN;
    42919:
        FuUnicodeCodepointCaseConvert := 42918;
        RETURN;
    42920:
        FuUnicodeCodepointCaseConvert := 42921;
        RETURN;
    42921:
        FuUnicodeCodepointCaseConvert := 42920;
        RETURN;
    42922:
        FuUnicodeCodepointCaseConvert := 614;
        RETURN;
    42923:
        FuUnicodeCodepointCaseConvert := 604;
        RETURN;
    42924:
        FuUnicodeCodepointCaseConvert := 609;
        RETURN;
    42925:
        FuUnicodeCodepointCaseConvert := 620;
        RETURN;
    42926:
        FuUnicodeCodepointCaseConvert := 618;
        RETURN;
    42928:
        FuUnicodeCodepointCaseConvert := 670;
        RETURN;
    42929:
        FuUnicodeCodepointCaseConvert := 647;
        RETURN;
    42930:
        FuUnicodeCodepointCaseConvert := 669;
        RETURN;
    42931:
        FuUnicodeCodepointCaseConvert := 43859;
        RETURN;
    42932:
        FuUnicodeCodepointCaseConvert := 42933;
        RETURN;
    42933:
        FuUnicodeCodepointCaseConvert := 42932;
        RETURN;
    42934:
        FuUnicodeCodepointCaseConvert := 42935;
        RETURN;
    42935:
        FuUnicodeCodepointCaseConvert := 42934;
        RETURN;
    42936:
        FuUnicodeCodepointCaseConvert := 42937;
        RETURN;
    42937:
        FuUnicodeCodepointCaseConvert := 42936;
        RETURN;
    42938:
        FuUnicodeCodepointCaseConvert := 42939;
        RETURN;
    42939:
        FuUnicodeCodepointCaseConvert := 42938;
        RETURN;
    42940:
        FuUnicodeCodepointCaseConvert := 42941;
        RETURN;
    42941:
        FuUnicodeCodepointCaseConvert := 42940;
        RETURN;
    42942:
        FuUnicodeCodepointCaseConvert := 42943;
        RETURN;
    42943:
        FuUnicodeCodepointCaseConvert := 42942;
        RETURN;
    42944:
        FuUnicodeCodepointCaseConvert := 42945;
        RETURN;
    42945:
        FuUnicodeCodepointCaseConvert := 42944;
        RETURN;
    42946:
        FuUnicodeCodepointCaseConvert := 42947;
        RETURN;
    42947:
        FuUnicodeCodepointCaseConvert := 42946;
        RETURN;
    42948:
        FuUnicodeCodepointCaseConvert := 42900;
        RETURN;
    42949:
        FuUnicodeCodepointCaseConvert := 642;
        RETURN;
    42950:
        FuUnicodeCodepointCaseConvert := 7566;
        RETURN;
    42951:
        FuUnicodeCodepointCaseConvert := 42952;
        RETURN;
    42952:
        FuUnicodeCodepointCaseConvert := 42951;
        RETURN;
    42953:
        FuUnicodeCodepointCaseConvert := 42954;
        RETURN;
    42954:
        FuUnicodeCodepointCaseConvert := 42953;
        RETURN;
    42960:
        FuUnicodeCodepointCaseConvert := 42961;
        RETURN;
    42961:
        FuUnicodeCodepointCaseConvert := 42960;
        RETURN;
    42966:
        FuUnicodeCodepointCaseConvert := 42967;
        RETURN;
    42967:
        FuUnicodeCodepointCaseConvert := 42966;
        RETURN;
    42968:
        FuUnicodeCodepointCaseConvert := 42969;
        RETURN;
    42969:
        FuUnicodeCodepointCaseConvert := 42968;
        RETURN;
    42997:
        FuUnicodeCodepointCaseConvert := 42998;
        RETURN;
    42998:
        FuUnicodeCodepointCaseConvert := 42997;
        RETURN;
    43859:
        FuUnicodeCodepointCaseConvert := 42931;
        RETURN;
    43888:
        FuUnicodeCodepointCaseConvert := 5024;
        RETURN;
    43889:
        FuUnicodeCodepointCaseConvert := 5025;
        RETURN;
    43890:
        FuUnicodeCodepointCaseConvert := 5026;
        RETURN;
    43891:
        FuUnicodeCodepointCaseConvert := 5027;
        RETURN;
    43892:
        FuUnicodeCodepointCaseConvert := 5028;
        RETURN;
    43893:
        FuUnicodeCodepointCaseConvert := 5029;
        RETURN;
    43894:
        FuUnicodeCodepointCaseConvert := 5030;
        RETURN;
    43895:
        FuUnicodeCodepointCaseConvert := 5031;
        RETURN;
    43896:
        FuUnicodeCodepointCaseConvert := 5032;
        RETURN;
    43897:
        FuUnicodeCodepointCaseConvert := 5033;
        RETURN;
    43898:
        FuUnicodeCodepointCaseConvert := 5034;
        RETURN;
    43899:
        FuUnicodeCodepointCaseConvert := 5035;
        RETURN;
    43900:
        FuUnicodeCodepointCaseConvert := 5036;
        RETURN;
    43901:
        FuUnicodeCodepointCaseConvert := 5037;
        RETURN;
    43902:
        FuUnicodeCodepointCaseConvert := 5038;
        RETURN;
    43903:
        FuUnicodeCodepointCaseConvert := 5039;
        RETURN;
    43904:
        FuUnicodeCodepointCaseConvert := 5040;
        RETURN;
    43905:
        FuUnicodeCodepointCaseConvert := 5041;
        RETURN;
    43906:
        FuUnicodeCodepointCaseConvert := 5042;
        RETURN;
    43907:
        FuUnicodeCodepointCaseConvert := 5043;
        RETURN;
    43908:
        FuUnicodeCodepointCaseConvert := 5044;
        RETURN;
    43909:
        FuUnicodeCodepointCaseConvert := 5045;
        RETURN;
    43910:
        FuUnicodeCodepointCaseConvert := 5046;
        RETURN;
    43911:
        FuUnicodeCodepointCaseConvert := 5047;
        RETURN;
    43912:
        FuUnicodeCodepointCaseConvert := 5048;
        RETURN;
    43913:
        FuUnicodeCodepointCaseConvert := 5049;
        RETURN;
    43914:
        FuUnicodeCodepointCaseConvert := 5050;
        RETURN;
    43915:
        FuUnicodeCodepointCaseConvert := 5051;
        RETURN;
    43916:
        FuUnicodeCodepointCaseConvert := 5052;
        RETURN;
    43917:
        FuUnicodeCodepointCaseConvert := 5053;
        RETURN;
    43918:
        FuUnicodeCodepointCaseConvert := 5054;
        RETURN;
    43919:
        FuUnicodeCodepointCaseConvert := 5055;
        RETURN;
    43920:
        FuUnicodeCodepointCaseConvert := 5056;
        RETURN;
    43921:
        FuUnicodeCodepointCaseConvert := 5057;
        RETURN;
    43922:
        FuUnicodeCodepointCaseConvert := 5058;
        RETURN;
    43923:
        FuUnicodeCodepointCaseConvert := 5059;
        RETURN;
    43924:
        FuUnicodeCodepointCaseConvert := 5060;
        RETURN;
    43925:
        FuUnicodeCodepointCaseConvert := 5061;
        RETURN;
    43926:
        FuUnicodeCodepointCaseConvert := 5062;
        RETURN;
    43927:
        FuUnicodeCodepointCaseConvert := 5063;
        RETURN;
    43928:
        FuUnicodeCodepointCaseConvert := 5064;
        RETURN;
    43929:
        FuUnicodeCodepointCaseConvert := 5065;
        RETURN;
    43930:
        FuUnicodeCodepointCaseConvert := 5066;
        RETURN;
    43931:
        FuUnicodeCodepointCaseConvert := 5067;
        RETURN;
    43932:
        FuUnicodeCodepointCaseConvert := 5068;
        RETURN;
    43933:
        FuUnicodeCodepointCaseConvert := 5069;
        RETURN;
    43934:
        FuUnicodeCodepointCaseConvert := 5070;
        RETURN;
    43935:
        FuUnicodeCodepointCaseConvert := 5071;
        RETURN;
    43936:
        FuUnicodeCodepointCaseConvert := 5072;
        RETURN;
    43937:
        FuUnicodeCodepointCaseConvert := 5073;
        RETURN;
    43938:
        FuUnicodeCodepointCaseConvert := 5074;
        RETURN;
    43939:
        FuUnicodeCodepointCaseConvert := 5075;
        RETURN;
    43940:
        FuUnicodeCodepointCaseConvert := 5076;
        RETURN;
    43941:
        FuUnicodeCodepointCaseConvert := 5077;
        RETURN;
    43942:
        FuUnicodeCodepointCaseConvert := 5078;
        RETURN;
    43943:
        FuUnicodeCodepointCaseConvert := 5079;
        RETURN;
    43944:
        FuUnicodeCodepointCaseConvert := 5080;
        RETURN;
    43945:
        FuUnicodeCodepointCaseConvert := 5081;
        RETURN;
    43946:
        FuUnicodeCodepointCaseConvert := 5082;
        RETURN;
    43947:
        FuUnicodeCodepointCaseConvert := 5083;
        RETURN;
    43948:
        FuUnicodeCodepointCaseConvert := 5084;
        RETURN;
    43949:
        FuUnicodeCodepointCaseConvert := 5085;
        RETURN;
    43950:
        FuUnicodeCodepointCaseConvert := 5086;
        RETURN;
    43951:
        FuUnicodeCodepointCaseConvert := 5087;
        RETURN;
    43952:
        FuUnicodeCodepointCaseConvert := 5088;
        RETURN;
    43953:
        FuUnicodeCodepointCaseConvert := 5089;
        RETURN;
    43954:
        FuUnicodeCodepointCaseConvert := 5090;
        RETURN;
    43955:
        FuUnicodeCodepointCaseConvert := 5091;
        RETURN;
    43956:
        FuUnicodeCodepointCaseConvert := 5092;
        RETURN;
    43957:
        FuUnicodeCodepointCaseConvert := 5093;
        RETURN;
    43958:
        FuUnicodeCodepointCaseConvert := 5094;
        RETURN;
    43959:
        FuUnicodeCodepointCaseConvert := 5095;
        RETURN;
    43960:
        FuUnicodeCodepointCaseConvert := 5096;
        RETURN;
    43961:
        FuUnicodeCodepointCaseConvert := 5097;
        RETURN;
    43962:
        FuUnicodeCodepointCaseConvert := 5098;
        RETURN;
    43963:
        FuUnicodeCodepointCaseConvert := 5099;
        RETURN;
    43964:
        FuUnicodeCodepointCaseConvert := 5100;
        RETURN;
    43965:
        FuUnicodeCodepointCaseConvert := 5101;
        RETURN;
    43966:
        FuUnicodeCodepointCaseConvert := 5102;
        RETURN;
    43967:
        FuUnicodeCodepointCaseConvert := 5103;
        RETURN;
    65313:
        FuUnicodeCodepointCaseConvert := 65345;
        RETURN;
    65314:
        FuUnicodeCodepointCaseConvert := 65346;
        RETURN;
    65315:
        FuUnicodeCodepointCaseConvert := 65347;
        RETURN;
    65316:
        FuUnicodeCodepointCaseConvert := 65348;
        RETURN;
    65317:
        FuUnicodeCodepointCaseConvert := 65349;
        RETURN;
    65318:
        FuUnicodeCodepointCaseConvert := 65350;
        RETURN;
    65319:
        FuUnicodeCodepointCaseConvert := 65351;
        RETURN;
    65320:
        FuUnicodeCodepointCaseConvert := 65352;
        RETURN;
    65321:
        FuUnicodeCodepointCaseConvert := 65353;
        RETURN;
    65322:
        FuUnicodeCodepointCaseConvert := 65354;
        RETURN;
    65323:
        FuUnicodeCodepointCaseConvert := 65355;
        RETURN;
    65324:
        FuUnicodeCodepointCaseConvert := 65356;
        RETURN;
    65325:
        FuUnicodeCodepointCaseConvert := 65357;
        RETURN;
    65326:
        FuUnicodeCodepointCaseConvert := 65358;
        RETURN;
    65327:
        FuUnicodeCodepointCaseConvert := 65359;
        RETURN;
    65328:
        FuUnicodeCodepointCaseConvert := 65360;
        RETURN;
    65329:
        FuUnicodeCodepointCaseConvert := 65361;
        RETURN;
    65330:
        FuUnicodeCodepointCaseConvert := 65362;
        RETURN;
    65331:
        FuUnicodeCodepointCaseConvert := 65363;
        RETURN;
    65332:
        FuUnicodeCodepointCaseConvert := 65364;
        RETURN;
    65333:
        FuUnicodeCodepointCaseConvert := 65365;
        RETURN;
    65334:
        FuUnicodeCodepointCaseConvert := 65366;
        RETURN;
    65335:
        FuUnicodeCodepointCaseConvert := 65367;
        RETURN;
    65336:
        FuUnicodeCodepointCaseConvert := 65368;
        RETURN;
    65337:
        FuUnicodeCodepointCaseConvert := 65369;
        RETURN;
    65338:
        FuUnicodeCodepointCaseConvert := 65370;
        RETURN;
    65345:
        FuUnicodeCodepointCaseConvert := 65313;
        RETURN;
    65346:
        FuUnicodeCodepointCaseConvert := 65314;
        RETURN;
    65347:
        FuUnicodeCodepointCaseConvert := 65315;
        RETURN;
    65348:
        FuUnicodeCodepointCaseConvert := 65316;
        RETURN;
    65349:
        FuUnicodeCodepointCaseConvert := 65317;
        RETURN;
    65350:
        FuUnicodeCodepointCaseConvert := 65318;
        RETURN;
    65351:
        FuUnicodeCodepointCaseConvert := 65319;
        RETURN;
    65352:
        FuUnicodeCodepointCaseConvert := 65320;
        RETURN;
    65353:
        FuUnicodeCodepointCaseConvert := 65321;
        RETURN;
    65354:
        FuUnicodeCodepointCaseConvert := 65322;
        RETURN;
    65355:
        FuUnicodeCodepointCaseConvert := 65323;
        RETURN;
    65356:
        FuUnicodeCodepointCaseConvert := 65324;
        RETURN;
    65357:
        FuUnicodeCodepointCaseConvert := 65325;
        RETURN;
    65358:
        FuUnicodeCodepointCaseConvert := 65326;
        RETURN;
    65359:
        FuUnicodeCodepointCaseConvert := 65327;
        RETURN;
    65360:
        FuUnicodeCodepointCaseConvert := 65328;
        RETURN;
    65361:
        FuUnicodeCodepointCaseConvert := 65329;
        RETURN;
    65362:
        FuUnicodeCodepointCaseConvert := 65330;
        RETURN;
    65363:
        FuUnicodeCodepointCaseConvert := 65331;
        RETURN;
    65364:
        FuUnicodeCodepointCaseConvert := 65332;
        RETURN;
    65365:
        FuUnicodeCodepointCaseConvert := 65333;
        RETURN;
    65366:
        FuUnicodeCodepointCaseConvert := 65334;
        RETURN;
    65367:
        FuUnicodeCodepointCaseConvert := 65335;
        RETURN;
    65368:
        FuUnicodeCodepointCaseConvert := 65336;
        RETURN;
    65369:
        FuUnicodeCodepointCaseConvert := 65337;
        RETURN;
    65370:
        FuUnicodeCodepointCaseConvert := 65338;
        RETURN;
    66560:
        FuUnicodeCodepointCaseConvert := 66600;
        RETURN;
    66561:
        FuUnicodeCodepointCaseConvert := 66601;
        RETURN;
    66562:
        FuUnicodeCodepointCaseConvert := 66602;
        RETURN;
    66563:
        FuUnicodeCodepointCaseConvert := 66603;
        RETURN;
    66564:
        FuUnicodeCodepointCaseConvert := 66604;
        RETURN;
    66565:
        FuUnicodeCodepointCaseConvert := 66605;
        RETURN;
    66566:
        FuUnicodeCodepointCaseConvert := 66606;
        RETURN;
    66567:
        FuUnicodeCodepointCaseConvert := 66607;
        RETURN;
    66568:
        FuUnicodeCodepointCaseConvert := 66608;
        RETURN;
    66569:
        FuUnicodeCodepointCaseConvert := 66609;
        RETURN;
    66570:
        FuUnicodeCodepointCaseConvert := 66610;
        RETURN;
    66571:
        FuUnicodeCodepointCaseConvert := 66611;
        RETURN;
    66572:
        FuUnicodeCodepointCaseConvert := 66612;
        RETURN;
    66573:
        FuUnicodeCodepointCaseConvert := 66613;
        RETURN;
    66574:
        FuUnicodeCodepointCaseConvert := 66614;
        RETURN;
    66575:
        FuUnicodeCodepointCaseConvert := 66615;
        RETURN;
    66576:
        FuUnicodeCodepointCaseConvert := 66616;
        RETURN;
    66577:
        FuUnicodeCodepointCaseConvert := 66617;
        RETURN;
    66578:
        FuUnicodeCodepointCaseConvert := 66618;
        RETURN;
    66579:
        FuUnicodeCodepointCaseConvert := 66619;
        RETURN;
    66580:
        FuUnicodeCodepointCaseConvert := 66620;
        RETURN;
    66581:
        FuUnicodeCodepointCaseConvert := 66621;
        RETURN;
    66582:
        FuUnicodeCodepointCaseConvert := 66622;
        RETURN;
    66583:
        FuUnicodeCodepointCaseConvert := 66623;
        RETURN;
    66584:
        FuUnicodeCodepointCaseConvert := 66624;
        RETURN;
    66585:
        FuUnicodeCodepointCaseConvert := 66625;
        RETURN;
    66586:
        FuUnicodeCodepointCaseConvert := 66626;
        RETURN;
    66587:
        FuUnicodeCodepointCaseConvert := 66627;
        RETURN;
    66588:
        FuUnicodeCodepointCaseConvert := 66628;
        RETURN;
    66589:
        FuUnicodeCodepointCaseConvert := 66629;
        RETURN;
    66590:
        FuUnicodeCodepointCaseConvert := 66630;
        RETURN;
    66591:
        FuUnicodeCodepointCaseConvert := 66631;
        RETURN;
    66592:
        FuUnicodeCodepointCaseConvert := 66632;
        RETURN;
    66593:
        FuUnicodeCodepointCaseConvert := 66633;
        RETURN;
    66594:
        FuUnicodeCodepointCaseConvert := 66634;
        RETURN;
    66595:
        FuUnicodeCodepointCaseConvert := 66635;
        RETURN;
    66596:
        FuUnicodeCodepointCaseConvert := 66636;
        RETURN;
    66597:
        FuUnicodeCodepointCaseConvert := 66637;
        RETURN;
    66598:
        FuUnicodeCodepointCaseConvert := 66638;
        RETURN;
    66599:
        FuUnicodeCodepointCaseConvert := 66639;
        RETURN;
    66600:
        FuUnicodeCodepointCaseConvert := 66560;
        RETURN;
    66601:
        FuUnicodeCodepointCaseConvert := 66561;
        RETURN;
    66602:
        FuUnicodeCodepointCaseConvert := 66562;
        RETURN;
    66603:
        FuUnicodeCodepointCaseConvert := 66563;
        RETURN;
    66604:
        FuUnicodeCodepointCaseConvert := 66564;
        RETURN;
    66605:
        FuUnicodeCodepointCaseConvert := 66565;
        RETURN;
    66606:
        FuUnicodeCodepointCaseConvert := 66566;
        RETURN;
    66607:
        FuUnicodeCodepointCaseConvert := 66567;
        RETURN;
    66608:
        FuUnicodeCodepointCaseConvert := 66568;
        RETURN;
    66609:
        FuUnicodeCodepointCaseConvert := 66569;
        RETURN;
    66610:
        FuUnicodeCodepointCaseConvert := 66570;
        RETURN;
    66611:
